C05487=1125.675,192.025,-64.166,-179.144,9.235,149.572
C05488=1125.671,192.273,-64.190,-179.142,9.238,149.572
C05489=1125.666,192.521,-64.214,-179.140,9.241,149.572
C05490=1125.662,192.771,-64.239,-179.138,9.243,149.572
C05491=1125.657,193.020,-64.262,-179.136,9.246,149.572
C05492=1125.652,193.269,-64.287,-179.135,9.248,149.572
C05493=1125.648,193.517,-64.311,-179.133,9.251,149.572
C05494=1125.644,193.766,-64.336,-179.131,9.254,149.573
C05495=1125.639,194.015,-64.360,-179.129,9.257,149.573
C05496=1125.634,194.263,-64.384,-179.127,9.259,149.573
C05497=1125.630,194.513,-64.409,-179.126,9.262,149.573
C05498=1125.625,194.761,-64.433,-179.124,9.264,149.573
C05499=1125.620,195.010,-64.458,-179.122,9.267,149.573
C05500=1125.616,195.259,-64.482,-179.121,9.269,149.573
C05501=1125.612,195.507,-64.508,-179.119,9.272,149.573
C05502=1125.607,195.755,-64.532,-179.117,9.274,149.574
C05503=1125.603,196.004,-64.556,-179.116,9.277,149.574
C05504=1125.598,196.253,-64.581,-179.114,9.279,149.574
C05505=1125.594,196.502,-64.605,-179.111,9.283,149.574
C05506=1125.589,196.751,-64.630,-179.107,9.287,149.574
C05507=1125.585,196.999,-64.654,-179.104,9.290,149.574
C05508=1125.580,197.248,-64.679,-179.099,9.295,149.574
C05509=1125.576,197.497,-64.703,-179.096,9.298,149.573
C05510=1125.571,197.745,-64.729,-179.092,9.302,149.573
C05511=1125.567,197.995,-64.754,-179.089,9.305,149.573
C05512=1125.562,198.209,-64.774,-179.086,9.308,149.573
C05513=1125.559,198.423,-64.796,-179.083,9.311,149.573
C05514=1125.555,198.637,-64.817,-179.080,9.315,149.573
C05515=1125.551,198.851,-64.839,-179.077,9.317,149.573
C05516=1125.547,199.065,-64.859,-179.074,9.320,149.573
C05517=1125.544,199.279,-64.881,-179.071,9.323,149.573
C05518=1125.540,199.492,-64.902,-179.068,9.326,149.573
C05519=1125.536,199.706,-64.923,-179.065,9.329,149.572
C05520=1125.531,199.956,-64.948,-179.062,9.332,149.572
C05521=1125.526,200.204,-64.973,-179.058,9.336,149.572
C05522=1125.523,200.453,-64.998,-179.055,9.339,149.572
C05523=1125.518,200.702,-65.023,-179.052,9.342,149.572
C05524=1125.513,200.951,-65.049,-179.048,9.345,149.572
C05525=1125.509,201.199,-65.073,-179.044,9.349,149.572
C05526=1125.505,201.448,-65.098,-179.042,9.352,149.571
C05527=1125.500,201.696,-65.123,-179.038,9.356,149.571
C05528=1125.496,201.946,-65.148,-179.035,9.358,149.571
C05529=1125.491,202.194,-65.173,-179.032,9.362,149.571
C05530=1125.487,202.443,-65.198,-179.029,9.365,149.571
C05531=1125.482,202.691,-65.223,-179.026,9.367,149.571
C05532=1125.478,202.940,-65.248,-179.022,9.371,149.571
C05533=1125.473,203.188,-65.273,-179.019,9.374,149.571
C05534=1125.469,203.438,-65.298,-179.016,9.376,149.570
C05535=1125.464,203.686,-65.324,-179.014,9.379,149.571
C05536=1125.459,203.935,-65.349,-179.010,9.383,149.570
C05537=1125.455,204.183,-65.374,-179.007,9.386,149.570
C05538=1125.451,204.432,-65.399,-179.004,9.388,149.570
C05539=1125.446,204.681,-65.424,-179.001,9.391,149.570
C05540=1125.442,204.929,-65.450,-178.999,9.394,149.570
C05541=1125.437,205.178,-65.475,-178.996,9.397,149.570
C05542=1125.432,205.427,-65.500,-178.993,9.400,149.570
C05543=1125.429,205.676,-65.525,-178.990,9.402,149.570
C05544=1125.424,205.924,-65.551,-178.988,9.406,149.570
C05545=1125.419,206.173,-65.576,-178.985,9.408,149.569
C05546=1125.415,206.422,-65.601,-178.982,9.411,149.569
C05547=1125.410,206.670,-65.627,-178.979,9.414,149.569
C05548=1125.406,206.919,-65.652,-178.976,9.417,149.569
C05549=1125.401,207.167,-65.677,-178.974,9.420,149.569
C05550=1125.397,207.416,-65.703,-178.971,9.422,149.569
C05551=1125.393,207.665,-65.729,-178.969,9.425,149.569
C05552=1125.387,207.914,-65.753,-178.966,9.428,149.569
C05553=1125.383,208.163,-65.779,-178.963,9.431,149.569
C05554=1125.379,208.411,-65.805,-178.961,9.433,149.569
C05555=1125.375,208.659,-65.830,-178.958,9.436,149.569
C05556=1125.371,208.908,-65.855,-178.956,9.439,149.569
C05557=1125.366,209.157,-65.881,-178.954,9.441,149.569
C05558=1125.361,209.406,-65.906,-178.951,9.444,149.569
C05559=1125.357,209.654,-65.932,-178.949,9.446,149.569
C05560=1125.353,209.903,-65.957,-178.947,9.450,149.569
C05561=1125.348,210.151,-65.983,-178.944,9.453,149.569
C05562=1125.344,210.400,-66.009,-178.942,9.455,149.569
C05563=1125.340,210.649,-66.034,-178.940,9.457,149.569
C05564=1125.334,210.897,-66.060,-178.937,9.460,149.569
C05565=1125.330,211.146,-66.086,-178.936,9.462,149.569
C05566=1125.326,211.395,-66.112,-178.933,9.466,149.569
C05567=1125.321,211.643,-66.137,-178.932,9.468,149.569
C05568=1125.317,211.857,-66.159,-178.930,9.471,149.569
C05569=1125.313,212.071,-66.181,-178.928,9.473,149.569
C05570=1125.310,212.285,-66.203,-178.926,9.475,149.570
C05571=1125.306,212.500,-66.225,-178.924,9.478,149.570
C05572=1125.302,212.713,-66.248,-178.923,9.480,149.570
C05573=1125.298,212.927,-66.270,-178.921,9.482,149.570
C05574=1125.295,213.140,-66.292,-178.919,9.484,149.570
C05575=1125.290,213.355,-66.314,-178.918,9.487,149.570
C05576=1125.286,213.604,-66.340,-178.916,9.489,149.570
C05577=1125.281,213.852,-66.365,-178.914,9.492,149.570
C05578=1125.277,214.100,-66.391,-178.912,9.495,149.571
C05579=1125.273,214.349,-66.416,-178.910,9.497,149.571
C05580=1125.269,214.598,-66.442,-178.909,9.500,149.571
C05581=1125.263,214.846,-66.468,-178.906,9.503,149.571
C05582=1125.259,215.095,-66.494,-178.905,9.506,149.571
C05583=1125.255,215.343,-66.520,-178.902,9.509,149.571
C05584=1125.251,215.592,-66.546,-178.900,9.511,149.571
C05585=1125.247,215.841,-66.572,-178.898,9.515,149.571
C05586=1125.242,216.089,-66.597,-178.896,9.517,149.572
C05587=1125.237,216.338,-66.624,-178.894,9.521,149.572
C05588=1125.233,216.587,-66.649,-178.892,9.523,149.572
C05589=1125.229,216.835,-66.676,-178.890,9.526,149.572
C05590=1125.224,217.084,-66.702,-178.888,9.529,149.572
C05591=1125.220,217.332,-66.727,-178.886,9.532,149.572
C05592=1125.215,217.581,-66.753,-178.883,9.535,149.572
C05593=1125.210,217.830,-66.779,-178.881,9.538,149.572
C05594=1125.206,218.078,-66.806,-178.879,9.541,149.573
C05595=1125.202,218.327,-66.831,-178.877,9.544,149.573
C05596=1125.198,218.576,-66.857,-178.874,9.547,149.573
C05597=1125.193,218.824,-66.884,-178.872,9.550,149.573
C05598=1125.189,219.073,-66.910,-178.869,9.554,149.573
C05599=1125.184,219.321,-66.935,-178.868,9.556,149.573
C05600=1125.179,219.570,-66.962,-178.865,9.559,149.573
C05601=1125.175,219.819,-66.988,-178.862,9.562,149.573
C05602=1125.171,220.067,-67.014,-178.860,9.565,149.573
C05603=1125.167,220.316,-67.040,-178.857,9.568,149.573
C05604=1125.162,220.564,-67.066,-178.855,9.571,149.573
C05605=1125.157,220.813,-67.092,-178.852,9.574,149.573
C05606=1125.154,221.061,-67.119,-178.850,9.578,149.573
C05607=1125.149,221.310,-67.145,-178.847,9.581,149.574
C05608=1125.144,221.559,-67.171,-178.845,9.584,149.574
C05609=1125.140,221.807,-67.198,-178.842,9.588,149.574
C05610=1125.135,222.056,-67.223,-178.839,9.591,149.574
C05611=1125.132,222.304,-67.250,-178.837,9.594,149.574
C05612=1125.127,222.554,-67.276,-178.834,9.597,149.574
C05613=1125.123,222.802,-67.303,-178.832,9.600,149.574
C05614=1125.118,223.050,-67.328,-178.828,9.604,149.574
C05615=1125.113,223.298,-67.355,-178.826,9.607,149.574
C05616=1125.109,223.547,-67.381,-178.823,9.610,149.574
C05617=1125.104,223.796,-67.408,-178.820,9.613,149.574
C05618=1125.100,224.044,-67.434,-178.817,9.617,149.574
C05619=1125.095,224.293,-67.461,-178.814,9.620,149.574
C05620=1125.092,224.541,-67.487,-178.811,9.624,149.574
C05621=1125.087,224.790,-67.514,-178.809,9.627,149.574
C05622=1125.083,225.038,-67.540,-178.806,9.629,149.574
C05623=1125.078,225.287,-67.567,-178.802,9.633,149.574
C05624=1125.075,225.500,-67.589,-178.800,9.636,149.574
C05625=1125.071,225.715,-67.612,-178.797,9.639,149.574
C05626=1125.067,225.928,-67.635,-178.795,9.641,149.574
C05627=1125.063,226.142,-67.658,-178.792,9.644,149.574
C05628=1125.059,226.356,-67.681,-178.790,9.647,149.574
C05629=1125.056,226.570,-67.704,-178.787,9.650,149.574
C05630=1125.052,226.784,-67.727,-178.784,9.653,149.574
C05631=1125.048,226.997,-67.750,-178.781,9.656,149.574
C05632=1125.044,227.245,-67.776,-178.778,9.659,149.574
C05633=1125.039,227.494,-67.802,-178.775,9.663,149.574
C05634=1125.034,227.743,-67.829,-178.772,9.666,149.574
C05635=1125.030,227.991,-67.856,-178.768,9.670,149.574
C05636=1125.026,228.240,-67.883,-178.765,9.672,149.573
C05637=1125.022,228.489,-67.910,-178.761,9.676,149.573
C05638=1125.017,228.738,-67.936,-178.758,9.680,149.573
C05639=1125.013,228.986,-67.963,-178.755,9.683,149.573
C05640=1125.009,229.234,-67.990,-178.752,9.686,149.573
C05641=1125.004,229.483,-68.017,-178.748,9.689,149.573
C05642=1124.999,229.731,-68.044,-178.745,9.693,149.573
C05643=1124.995,229.980,-68.070,-178.741,9.696,149.573
C05644=1124.991,230.228,-68.097,-178.737,9.700,149.572
C05645=1124.986,230.477,-68.124,-178.734,9.702,149.572
C05646=1124.982,230.725,-68.151,-178.730,9.706,149.572
C05647=1124.978,230.974,-68.178,-178.727,9.709,149.572
C05648=1124.973,231.222,-68.205,-178.724,9.712,149.572
C05649=1124.969,231.471,-68.232,-178.720,9.716,149.572
C05650=1124.965,231.719,-68.259,-178.717,9.719,149.572
C05651=1124.960,231.968,-68.286,-178.714,9.722,149.572
C05652=1124.956,232.216,-68.313,-178.711,9.725,149.571
C05653=1124.951,232.465,-68.340,-178.707,9.728,149.571
C05654=1124.947,232.714,-68.367,-178.704,9.731,149.571
C05655=1124.943,232.962,-68.394,-178.701,9.733,149.571
C05656=1124.939,233.210,-68.422,-178.697,9.737,149.571
C05657=1124.934,233.458,-68.449,-178.694,9.740,149.571
C05658=1124.930,233.708,-68.476,-178.691,9.742,149.571
C05659=1124.925,233.956,-68.503,-178.689,9.745,149.570
C05660=1124.921,234.205,-68.530,-178.685,9.749,149.570
C05661=1124.917,234.452,-68.558,-178.682,9.751,149.570
C05662=1124.912,234.701,-68.585,-178.679,9.754,149.570
C05663=1124.908,234.950,-68.612,-178.676,9.757,149.570
C05664=1124.904,235.198,-68.639,-178.673,9.760,149.570
C05665=1124.899,235.447,-68.666,-178.670,9.762,149.570
C05666=1124.895,235.695,-68.694,-178.668,9.766,149.570
C05667=1124.890,235.944,-68.721,-178.665,9.768,149.570
C05668=1124.886,236.192,-68.748,-178.662,9.771,149.570
C05669=1124.881,236.440,-68.776,-178.659,9.773,149.569
C05670=1124.877,236.689,-68.803,-178.657,9.776,149.569
C05671=1124.873,236.938,-68.831,-178.654,9.779,149.569
C05672=1124.868,237.186,-68.858,-178.651,9.781,149.569
C05673=1124.864,237.434,-68.886,-178.649,9.784,149.569
C05674=1124.861,237.683,-68.913,-178.646,9.786,149.569
C05675=1124.856,237.931,-68.940,-178.643,9.789,149.569
C05676=1124.851,238.180,-68.967,-178.641,9.791,149.569
C05677=1124.847,238.427,-68.995,-178.638,9.794,149.569
C05678=1124.842,238.677,-69.023,-178.635,9.797,149.569
C05679=1124.838,238.925,-69.051,-178.633,9.799,149.568
C05680=1124.835,239.139,-69.074,-178.631,9.801,149.569
C05681=1124.831,239.352,-69.097,-178.629,9.803,149.568
C05682=1124.828,239.566,-69.121,-178.626,9.805,149.568
C05683=1124.823,239.779,-69.145,-178.624,9.808,149.568
C05684=1124.820,239.994,-69.169,-178.622,9.810,149.568
C05685=1124.816,240.207,-69.192,-178.620,9.812,149.568
C05686=1124.812,240.421,-69.217,-178.618,9.814,149.568
C05687=1124.808,240.634,-69.240,-178.616,9.816,149.568
C05688=1124.804,240.883,-69.267,-178.614,9.818,149.568
C05689=1124.800,241.131,-69.295,-178.612,9.820,149.568
C05690=1124.795,241.379,-69.322,-178.609,9.824,149.568
C05691=1124.792,241.628,-69.350,-178.607,9.826,149.568
C05692=1124.786,241.877,-69.378,-178.605,9.828,149.568
C05693=1124.782,242.124,-69.406,-178.603,9.830,149.568
C05694=1124.778,242.373,-69.434,-178.601,9.833,149.568
C05695=1124.773,242.622,-69.461,-178.599,9.834,149.568
C05696=1124.770,242.870,-69.489,-178.596,9.838,149.568
C05697=1124.765,243.119,-69.516,-178.594,9.840,149.568
C05698=1124.761,243.367,-69.544,-178.593,9.842,149.568
C05699=1124.756,243.615,-69.573,-178.591,9.845,149.568
C05700=1124.752,243.864,-69.600,-178.589,9.847,149.568
C05701=1124.748,244.112,-69.628,-178.587,9.849,149.568
C05702=1124.743,244.360,-69.656,-178.585,9.852,149.568
C05703=1124.739,244.609,-69.683,-178.584,9.853,149.568
C05704=1124.735,244.857,-69.711,-178.582,9.855,149.569
C05705=1124.730,245.106,-69.739,-178.580,9.858,149.569
C05706=1124.726,245.354,-69.767,-178.578,9.860,149.569
C05707=1124.722,245.603,-69.795,-178.576,9.862,149.569
C05708=1124.717,245.851,-69.822,-178.575,9.865,149.569
C05709=1124.713,246.099,-69.850,-178.573,9.867,149.569
C05710=1124.708,246.347,-69.879,-178.571,9.869,149.569
C05711=1124.704,246.597,-69.906,-178.570,9.872,149.569
C05712=1124.700,246.844,-69.934,-178.568,9.874,149.569
C05713=1124.696,247.093,-69.962,-178.567,9.876,149.570
C05714=1124.691,247.341,-69.991,-178.565,9.878,149.570
C05715=1124.687,247.590,-70.019,-178.561,9.883,149.570
C05716=1124.683,247.838,-70.046,-178.555,9.887,149.569
C05717=1124.679,248.087,-70.074,-178.549,9.892,149.569
C05718=1124.674,248.335,-70.102,-178.544,9.897,149.568
C05719=1124.670,248.584,-70.130,-178.537,9.902,149.568
C05720=1124.666,248.831,-70.158,-178.532,9.906,149.567
C05721=1124.661,249.080,-70.187,-178.526,9.910,149.567
C05722=1124.657,249.328,-70.215,-178.521,9.914,149.567
C05723=1124.652,249.577,-70.243,-178.516,9.918,149.566
C05724=1124.648,249.825,-70.271,-178.512,9.922,149.566
C05725=1124.644,250.074,-70.299,-178.507,9.925,149.565
C05726=1124.639,250.322,-70.328,-178.503,9.929,149.565
C05727=1124.635,250.570,-70.356,-178.499,9.932,149.565
C05728=1124.630,250.818,-70.384,-178.495,9.935,149.565
C05729=1124.627,251.067,-70.412,-178.491,9.938,149.564
C05730=1124.622,251.315,-70.442,-178.487,9.941,149.564
C05731=1124.618,251.563,-70.470,-178.484,9.944,149.564
C05732=1124.614,251.812,-70.498,-178.480,9.946,149.564
C05733=1124.609,252.060,-70.526,-178.477,9.949,149.563
C05734=1124.606,252.309,-70.554,-178.474,9.952,149.563
C05735=1124.601,252.557,-70.583,-178.471,9.954,149.563
C05736=1124.597,252.770,-70.608,-178.469,9.956,149.563
C05737=1124.594,252.984,-70.632,-178.467,9.958,149.563
C05738=1124.590,253.197,-70.657,-178.465,9.960,149.563
C05739=1124.586,253.411,-70.681,-178.464,9.961,149.563
C05740=1124.582,253.624,-70.706,-178.462,9.963,149.563
C05741=1124.579,253.838,-70.730,-178.461,9.964,149.563
C05742=1124.575,254.052,-70.755,-178.460,9.966,149.563
C05743=1124.572,254.265,-70.780,-178.458,9.967,149.563
C05744=1124.567,254.513,-70.807,-178.457,9.969,149.563
C05745=1124.563,254.762,-70.836,-178.456,9.970,149.563
C05746=1124.559,255.010,-70.866,-178.456,9.972,149.563
C05747=1124.554,255.258,-70.893,-178.455,9.973,149.563
C05748=1124.550,255.507,-70.922,-178.455,9.974,149.564
C05749=1124.546,255.755,-70.951,-178.455,9.975,149.564
C05750=1124.541,256.003,-70.979,-178.455,9.976,149.564
C05751=1124.537,256.252,-71.008,-178.452,9.979,149.564
C05752=1124.533,256.500,-71.037,-178.449,9.982,149.564
C05753=1124.528,256.748,-71.065,-178.446,9.985,149.564
C05754=1124.524,256.997,-71.094,-178.443,9.987,149.564
C05755=1124.520,257.245,-71.123,-178.441,9.990,149.564
C05756=1124.516,257.493,-71.151,-178.437,9.994,149.564
C05757=1124.511,257.742,-71.179,-178.434,9.997,149.563
C05758=1124.507,257.990,-71.209,-178.431,9.999,149.563
C05759=1124.503,258.238,-71.237,-178.428,10.002,149.563
C05760=1124.499,258.486,-71.266,-178.425,10.005,149.563
C05761=1124.494,258.735,-71.295,-178.422,10.008,149.563
C05762=1124.491,258.983,-71.324,-178.419,10.011,149.563
C05763=1124.486,259.231,-71.352,-178.416,10.014,149.563
C05764=1124.481,259.480,-71.382,-178.413,10.017,149.563
C05765=1124.478,259.728,-71.410,-178.410,10.019,149.563
C05766=1124.474,259.976,-71.439,-178.406,10.023,149.562
C05767=1124.468,260.225,-71.468,-178.403,10.026,149.562
C05768=1124.464,260.473,-71.497,-178.400,10.028,149.562
C05769=1124.461,260.721,-71.525,-178.397,10.032,149.562
C05770=1124.456,260.970,-71.555,-178.393,10.034,149.562
C05771=1124.452,261.217,-71.584,-178.390,10.038,149.562
C05772=1124.447,261.466,-71.612,-178.387,10.041,149.562
C05773=1124.444,261.714,-71.641,-178.384,10.043,149.561
C05774=1124.439,261.963,-71.670,-178.380,10.047,149.561
C05775=1124.435,262.211,-71.699,-178.377,10.049,149.561
C05776=1124.430,262.459,-71.729,-178.373,10.052,149.561
C05777=1124.426,262.707,-71.758,-178.370,10.055,149.561
C05778=1124.422,262.956,-71.787,-178.366,10.058,149.561
C05779=1124.418,263.204,-71.816,-178.363,10.062,149.560
C05780=1124.414,263.452,-71.845,-178.359,10.064,149.560
C05781=1124.409,263.700,-71.874,-178.355,10.068,149.560
C05782=1124.405,263.949,-71.903,-178.352,10.070,149.560
C05783=1124.400,264.197,-71.932,-178.348,10.073,149.559
C05784=1124.396,264.445,-71.962,-178.344,10.077,149.559
C05785=1124.392,264.693,-71.991,-178.342,10.079,149.559
C05786=1124.388,264.942,-72.021,-178.339,10.081,149.559
C05787=1124.383,265.191,-72.049,-178.337,10.083,149.559
C05788=1124.379,265.438,-72.079,-178.334,10.086,149.559
C05789=1124.374,265.686,-72.108,-178.332,10.088,149.559
C05790=1124.370,265.935,-72.137,-178.329,10.091,149.559
C05791=1124.366,266.183,-72.167,-178.327,10.093,149.559
C05792=1124.363,266.396,-72.192,-178.324,10.095,149.558
C05793=1124.359,266.610,-72.217,-178.322,10.097,149.558
C05794=1124.355,266.823,-72.242,-178.320,10.099,149.558
C05795=1124.352,267.037,-72.268,-178.318,10.101,149.558
C05796=1124.348,267.250,-72.293,-178.316,10.103,149.558
C05797=1124.345,267.463,-72.318,-178.313,10.105,149.558
C05798=1124.341,267.677,-72.343,-178.310,10.108,149.558
C05799=1124.338,267.890,-72.368,-178.308,10.110,149.558
C05800=1124.333,268.139,-72.398,-178.306,10.112,149.558
C05801=1124.329,268.387,-72.427,-178.303,10.115,149.558
C05802=1124.325,268.635,-72.457,-178.300,10.118,149.558
C05803=1124.320,268.884,-72.487,-178.298,10.120,149.558
C05804=1124.316,269.132,-72.516,-178.295,10.123,149.557
C05805=1124.311,269.380,-72.545,-178.292,10.126,149.557
C05806=1124.307,269.627,-72.575,-178.290,10.127,149.557
C05807=1124.303,269.875,-72.605,-178.287,10.130,149.557
C05808=1124.299,270.124,-72.634,-178.284,10.133,149.557
C05809=1124.295,270.372,-72.664,-178.281,10.136,149.557
C05810=1124.291,270.620,-72.693,-178.279,10.138,149.557
C05811=1124.286,270.869,-72.723,-178.276,10.141,149.557
C05812=1124.282,271.117,-72.752,-178.273,10.143,149.557
C05813=1124.278,271.365,-72.782,-178.270,10.146,149.556
C05814=1124.273,271.613,-72.812,-178.267,10.149,149.556
C05815=1124.269,271.861,-72.842,-178.264,10.151,149.556
C05816=1124.265,272.110,-72.871,-178.261,10.153,149.556
C05817=1124.261,272.358,-72.901,-178.258,10.156,149.556
C05818=1124.257,272.606,-72.930,-178.255,10.159,149.556
C05819=1124.253,272.854,-72.960,-178.252,10.161,149.556
C05820=1124.248,273.102,-72.990,-178.249,10.164,149.556
C05821=1124.244,273.351,-73.020,-178.247,10.167,149.555
C05822=1124.240,273.599,-73.050,-178.244,10.170,149.555
C05823=1124.236,273.847,-73.080,-178.241,10.172,149.555
C05824=1124.232,274.095,-73.109,-178.237,10.175,149.555
C05825=1124.227,274.343,-73.140,-178.234,10.178,149.555
C05826=1124.223,274.592,-73.170,-178.231,10.180,149.555
C05827=1124.219,274.840,-73.199,-178.228,10.183,149.555
C05828=1124.215,275.088,-73.229,-178.226,10.186,149.555
C05829=1124.210,275.336,-73.259,-178.222,10.188,149.554
C05830=1124.206,275.584,-73.289,-178.219,10.191,149.554
C05831=1124.202,275.832,-73.319,-178.216,10.194,149.554
C05832=1124.198,276.080,-73.348,-178.213,10.197,149.554
C05833=1124.193,276.328,-73.379,-178.210,10.199,149.554
C05834=1124.190,276.577,-73.409,-178.207,10.202,149.554
C05835=1124.186,276.825,-73.439,-178.204,10.205,149.553
C05836=1124.181,277.074,-73.469,-178.200,10.208,149.553
C05837=1124.177,277.321,-73.499,-178.197,10.211,149.553
C05838=1124.173,277.569,-73.529,-178.194,10.213,149.553
C05839=1124.168,277.817,-73.559,-178.191,10.216,149.553
C05840=1124.164,278.066,-73.589,-178.188,10.218,149.553
C05841=1124.161,278.314,-73.619,-178.185,10.221,149.552
C05842=1124.156,278.563,-73.650,-178.181,10.224,149.552
C05843=1124.152,278.810,-73.680,-178.178,10.227,149.552
C05844=1124.148,279.058,-73.710,-178.175,10.230,149.552
C05845=1124.143,279.306,-73.740,-178.171,10.232,149.552
C05846=1124.139,279.554,-73.770,-178.169,10.235,149.552
C05847=1124.135,279.803,-73.801,-178.165,10.238,149.551
C05848=1124.132,280.016,-73.826,-178.162,10.240,149.551
C05849=1124.128,280.229,-73.853,-178.159,10.242,149.551
C05850=1124.125,280.442,-73.879,-178.156,10.245,149.551
C05851=1124.120,280.656,-73.905,-178.154,10.247,149.551
C05852=1124.118,280.869,-73.931,-178.150,10.249,149.550
C05853=1124.114,281.082,-73.957,-178.147,10.252,149.550
C05854=1124.110,281.296,-73.982,-178.144,10.255,149.550
C05855=1124.106,281.509,-74.009,-178.142,10.257,149.550
C05856=1124.102,281.757,-74.039,-178.138,10.259,149.550
C05857=1124.098,282.005,-74.070,-178.135,10.262,149.549
C05858=1124.094,282.253,-74.100,-178.133,10.265,149.549
C05859=1124.089,282.502,-74.130,-178.129,10.267,149.549
C05860=1124.085,282.749,-74.161,-178.126,10.270,149.549
C05861=1124.082,282.998,-74.192,-178.123,10.272,149.549
C05862=1124.077,283.246,-74.223,-178.120,10.275,149.549
C05863=1124.073,283.493,-74.253,-178.118,10.277,149.549
C05864=1124.068,283.741,-74.283,-178.114,10.279,149.548
C05865=1124.065,283.990,-74.314,-178.111,10.282,149.548
C05866=1124.061,284.238,-74.345,-178.108,10.285,149.548
C05867=1124.056,284.486,-74.375,-178.105,10.287,149.548
C05868=1124.052,284.735,-74.405,-178.102,10.290,149.547
C05869=1124.048,284.983,-74.436,-178.099,10.292,149.547
C05870=1124.043,285.231,-74.467,-178.096,10.295,149.547
C05871=1124.039,285.478,-74.497,-178.093,10.298,149.547
C05872=1124.035,285.727,-74.528,-178.090,10.300,149.547
C05873=1124.031,285.975,-74.559,-178.087,10.302,149.547
C05874=1124.027,286.222,-74.589,-178.084,10.305,149.547
C05875=1124.023,286.471,-74.620,-178.081,10.307,149.546
C05876=1124.018,286.719,-74.651,-178.078,10.310,149.546
C05877=1124.014,286.967,-74.681,-178.075,10.313,149.546
C05878=1124.011,287.215,-74.713,-178.071,10.315,149.546
C05879=1124.006,287.463,-74.744,-178.068,10.318,149.546
C05880=1124.003,287.711,-74.774,-178.065,10.320,149.545
C05881=1123.998,287.959,-74.805,-178.062,10.323,149.545
C05882=1123.993,288.207,-74.836,-178.059,10.325,149.545
C05883=1123.989,288.456,-74.867,-178.057,10.328,149.545
C05884=1123.986,288.703,-74.897,-178.053,10.330,149.545
C05885=1123.981,288.951,-74.928,-178.050,10.333,149.545
C05886=1123.977,289.199,-74.960,-178.047,10.335,149.544
C05887=1123.973,289.447,-74.991,-178.044,10.338,149.544
C05888=1123.969,289.696,-75.021,-178.041,10.341,149.544
C05889=1123.965,289.944,-75.052,-178.038,10.343,149.544
C05890=1123.960,290.191,-75.083,-178.035,10.346,149.544
C05891=1123.956,290.440,-75.114,-178.031,10.348,149.543
C05892=1123.952,290.687,-75.145,-178.029,10.351,149.543
C05893=1123.948,290.936,-75.176,-178.026,10.353,149.543
C05894=1123.944,291.183,-75.207,-178.023,10.355,149.543
C05895=1123.940,291.432,-75.238,-178.020,10.358,149.543
C05896=1123.936,291.680,-75.269,-178.017,10.361,149.543
C05897=1123.932,291.928,-75.301,-178.013,10.363,149.542
C05898=1123.927,292.176,-75.332,-178.010,10.366,149.542
C05899=1123.923,292.424,-75.363,-178.007,10.369,149.542
C05900=1123.919,292.672,-75.394,-178.004,10.371,149.542
C05901=1123.916,292.920,-75.425,-178.001,10.374,149.542
C05902=1123.911,293.167,-75.456,-177.998,10.376,149.542
C05903=1123.907,293.415,-75.487,-177.995,10.378,149.541
C05904=1123.903,293.629,-75.514,-177.992,10.381,149.541
C05905=1123.900,293.842,-75.541,-177.990,10.383,149.541
C05906=1123.896,294.056,-75.568,-177.987,10.385,149.541
C05907=1123.893,294.268,-75.595,-177.985,10.387,149.541
C05908=1123.889,294.482,-75.622,-177.982,10.389,149.541
C05909=1123.885,294.695,-75.649,-177.979,10.392,149.540
C05910=1123.882,294.907,-75.675,-177.977,10.394,149.540
C05911=1123.879,295.121,-75.702,-177.974,10.395,149.540
C05912=1123.875,295.368,-75.734,-177.971,10.398,149.540
C05913=1123.870,295.617,-75.765,-177.968,10.401,149.540
C05914=1123.867,295.865,-75.797,-177.965,10.403,149.540
C05915=1123.862,296.112,-75.828,-177.962,10.406,149.540
C05916=1123.858,296.361,-75.859,-177.958,10.409,149.539
C05917=1123.854,296.608,-75.891,-177.956,10.411,149.539
C05918=1123.849,296.857,-75.922,-177.952,10.414,149.539
C05919=1123.845,297.105,-75.954,-177.949,10.417,149.539
C05920=1123.841,297.353,-75.986,-177.946,10.419,149.539
C05921=1123.837,297.601,-76.016,-177.944,10.421,149.538
C05922=1123.833,297.849,-76.048,-177.940,10.423,149.538
C05923=1123.829,298.097,-76.080,-177.937,10.426,149.538
C05924=1123.825,298.345,-76.111,-177.934,10.429,149.538
C05925=1123.821,298.593,-76.143,-177.931,10.431,149.538
C05926=1123.817,298.840,-76.174,-177.928,10.434,149.537
C05927=1123.813,299.088,-76.206,-177.925,10.437,149.537
C05928=1123.809,299.337,-76.237,-177.922,10.439,149.537
C05929=1123.804,299.584,-76.269,-177.919,10.442,149.537
C05930=1123.800,299.832,-76.301,-177.915,10.444,149.537
C05931=1123.797,300.080,-76.333,-177.912,10.447,149.537
C05932=1123.792,300.328,-76.364,-177.910,10.449,149.536
C05933=1123.788,300.576,-76.396,-177.907,10.451,149.536
C05934=1123.784,300.824,-76.427,-177.903,10.454,149.536
C05935=1123.779,301.072,-76.459,-177.900,10.457,149.536
C05936=1123.776,301.320,-76.491,-177.897,10.459,149.536
C05937=1123.771,301.567,-76.523,-177.894,10.462,149.536
C05938=1123.768,301.816,-76.555,-177.891,10.464,149.535
C05939=1123.763,302.064,-76.587,-177.887,10.467,149.535
C05940=1123.759,302.311,-76.619,-177.885,10.469,149.535
C05941=1123.755,302.560,-76.650,-177.881,10.472,149.535
C05942=1123.751,302.808,-76.682,-177.878,10.475,149.535
C05943=1123.746,303.056,-76.714,-177.875,10.477,149.534
C05944=1123.743,303.304,-76.745,-177.873,10.479,149.534
C05945=1123.739,303.552,-76.777,-177.869,10.481,149.534
C05946=1123.734,303.799,-76.809,-177.866,10.484,149.534
C05947=1123.730,304.047,-76.841,-177.863,10.487,149.534
C05948=1123.726,304.295,-76.873,-177.860,10.489,149.534
C05949=1123.722,304.543,-76.906,-177.857,10.492,149.533
C05950=1123.718,304.790,-76.938,-177.854,10.495,149.533
C05951=1123.714,305.038,-76.970,-177.851,10.497,149.533
C05952=1123.710,305.287,-77.002,-177.848,10.500,149.533
C05953=1123.706,305.535,-77.034,-177.844,10.502,149.533
C05954=1123.702,305.782,-77.065,-177.841,10.505,149.533
C05955=1123.697,306.031,-77.098,-177.838,10.507,149.532
C05956=1123.694,306.279,-77.130,-177.835,10.510,149.532
C05957=1123.689,306.527,-77.162,-177.832,10.512,149.532
C05958=1123.685,306.774,-77.194,-177.829,10.514,149.532
C05959=1123.681,307.022,-77.226,-177.826,10.517,149.532
C05960=1123.678,307.235,-77.254,-177.823,10.519,149.531
C05961=1123.674,307.448,-77.281,-177.820,10.521,149.531
C05962=1123.671,307.661,-77.309,-177.818,10.523,149.531
C05963=1123.667,307.874,-77.337,-177.815,10.526,149.531
C05964=1123.663,308.087,-77.364,-177.813,10.528,149.531
C05965=1123.660,308.300,-77.392,-177.810,10.531,149.531
C05966=1123.656,308.514,-77.420,-177.807,10.532,149.530
C05967=1123.653,308.726,-77.447,-177.805,10.534,149.530
C05968=1123.649,308.973,-77.480,-177.802,10.537,149.530
C05969=1123.645,309.222,-77.512,-177.798,10.540,149.530
C05970=1123.641,309.470,-77.544,-177.795,10.542,149.530
C05971=1123.637,309.718,-77.577,-177.792,10.545,149.530
C05972=1123.633,309.965,-77.609,-177.789,10.547,149.529
C05973=1123.629,310.213,-77.642,-177.786,10.550,149.529
C05974=1123.625,310.461,-77.674,-177.783,10.552,149.529
C05975=1123.620,310.709,-77.706,-177.780,10.555,149.529
C05976=1123.617,310.956,-77.739,-177.776,10.558,149.529
C05977=1123.613,311.205,-77.771,-177.774,10.559,149.528
C05978=1123.608,311.453,-77.804,-177.771,10.562,149.528
C05979=1123.604,311.700,-77.836,-177.767,10.564,149.528
C05980=1123.600,311.948,-77.869,-177.764,10.567,149.528
C05981=1123.596,312.196,-77.901,-177.761,10.570,149.528
C05982=1123.592,312.443,-77.934,-177.758,10.572,149.528
C05983=1123.588,312.692,-77.967,-177.755,10.575,149.527
C05984=1123.584,312.939,-77.999,-177.751,10.577,149.527
C05985=1123.580,313.187,-78.032,-177.749,10.580,149.527
C05986=1123.577,313.435,-78.064,-177.745,10.583,149.527
C05987=1123.572,313.683,-78.097,-177.742,10.585,149.527
C05988=1123.568,313.931,-78.130,-177.739,10.588,149.527
C05989=1123.565,314.178,-78.162,-177.736,10.590,149.526
C05990=1123.560,314.427,-78.195,-177.733,10.593,149.526
C05991=1123.555,314.674,-78.227,-177.730,10.595,149.526
C05992=1123.552,314.922,-78.259,-177.727,10.597,149.526
C05993=1123.547,315.170,-78.292,-177.724,10.600,149.526
C05994=1123.543,315.417,-78.326,-177.720,10.602,149.525
C05995=1123.540,315.665,-78.357,-177.717,10.605,149.525
C05996=1123.536,315.913,-78.391,-177.714,10.607,149.525
C05997=1123.531,316.161,-78.424,-177.711,10.610,149.525
C05998=1123.527,316.409,-78.457,-177.708,10.613,149.525
C05999=1123.524,316.657,-78.489,-177.705,10.615,149.524
C06000=1123.519,316.904,-78.522,-177.702,10.618,149.524
C06001=1123.515,317.152,-78.555,-177.698,10.620,149.524
C06002=1123.511,317.400,-78.588,-177.695,10.623,149.524
C06003=1123.508,317.647,-78.621,-177.692,10.626,149.524
C06004=1123.503,317.896,-78.653,-177.689,10.628,149.524
C06005=1123.499,318.143,-78.686,-177.686,10.630,149.523
C06006=1123.495,318.391,-78.720,-177.683,10.632,149.523
C06007=1123.491,318.639,-78.753,-177.680,10.635,149.523
C06008=1123.488,318.887,-78.786,-177.677,10.638,149.523
C06009=1123.484,319.135,-78.819,-177.674,10.640,149.523
C06010=1123.480,319.382,-78.852,-177.670,10.643,149.522
C06011=1123.475,319.631,-78.884,-177.667,10.645,149.522
C06012=1123.471,319.878,-78.918,-177.664,10.648,149.522
C06013=1123.467,320.126,-78.951,-177.661,10.651,149.522
C06014=1123.463,320.374,-78.984,-177.658,10.653,149.522
C06015=1123.460,320.621,-79.016,-177.654,10.655,149.521
C06016=1123.456,320.834,-79.045,-177.652,10.657,149.521
C06017=1123.452,321.047,-79.074,-177.649,10.660,149.521
C06018=1123.450,321.260,-79.102,-177.646,10.662,149.521
C06019=1123.446,321.473,-79.131,-177.644,10.664,149.521
C06020=1123.442,321.685,-79.159,-177.641,10.666,149.521
C06021=1123.439,321.898,-79.187,-177.639,10.668,149.521
C06022=1123.435,322.111,-79.216,-177.636,10.670,149.520
C06023=1123.432,322.324,-79.245,-177.633,10.673,149.520
C06024=1123.428,322.571,-79.278,-177.630,10.675,149.520
C06025=1123.424,322.819,-79.312,-177.627,10.678,149.520
C06026=1123.420,323.067,-79.345,-177.623,10.680,149.520
C06027=1123.416,323.315,-79.378,-177.620,10.683,149.519
C06028=1123.412,323.563,-79.411,-177.618,10.685,149.519
C06029=1123.408,323.811,-79.445,-177.614,10.687,149.519
C06030=1123.404,324.058,-79.478,-177.611,10.690,149.519
C06031=1123.400,324.305,-79.512,-177.608,10.693,149.519
C06032=1123.396,324.553,-79.545,-177.605,10.695,149.519
C06033=1123.392,324.802,-79.578,-177.602,10.697,149.518
C06034=1123.388,325.049,-79.611,-177.599,10.700,149.518
C06035=1123.384,325.296,-79.645,-177.595,10.703,149.518
C06036=1123.380,325.544,-79.678,-177.592,10.705,149.518
C06037=1123.376,325.792,-79.712,-177.589,10.708,149.518
C06038=1123.372,326.040,-79.745,-177.586,10.710,149.517
C06039=1123.368,326.287,-79.779,-177.582,10.713,149.517
C06040=1123.364,326.535,-79.812,-177.579,10.716,149.517
C06041=1123.360,326.783,-79.845,-177.576,10.718,149.517
C06042=1123.356,327.030,-79.879,-177.573,10.720,149.517
C06043=1123.352,327.279,-79.913,-177.571,10.722,149.517
C06044=1123.348,327.527,-79.946,-177.567,10.725,149.516
C06045=1123.344,327.774,-79.980,-177.564,10.727,149.516
C06046=1123.340,328.021,-80.013,-177.561,10.730,149.516
C06047=1123.336,328.268,-80.047,-177.558,10.733,149.516
C06048=1123.333,328.517,-80.081,-177.554,10.735,149.516
C06049=1123.328,328.765,-80.115,-177.551,10.737,149.515
C06050=1123.324,329.012,-80.148,-177.548,10.740,149.515
C06051=1123.320,329.260,-80.182,-177.545,10.743,149.515
C06052=1123.317,329.508,-80.216,-177.541,10.745,149.515
C06053=1123.312,329.755,-80.249,-177.539,10.748,149.515
C06054=1123.308,330.003,-80.283,-177.535,10.750,149.514
C06055=1123.304,330.251,-80.317,-177.532,10.753,149.514
C06056=1123.300,330.498,-80.351,-177.529,10.755,149.514
C06057=1123.297,330.745,-80.385,-177.526,10.758,149.514
C06058=1123.292,330.993,-80.418,-177.522,10.760,149.514
C06059=1123.288,331.241,-80.453,-177.520,10.762,149.513
C06060=1123.284,331.489,-80.486,-177.517,10.765,149.513
C06061=1123.281,331.736,-80.520,-177.513,10.767,149.513
C06062=1123.277,331.984,-80.555,-177.510,10.770,149.513
C06063=1123.272,332.232,-80.588,-177.507,10.772,149.513
C06064=1123.269,332.479,-80.622,-177.504,10.775,149.513
C06065=1123.264,332.728,-80.656,-177.501,10.777,149.512
C06066=1123.260,332.975,-80.690,-177.497,10.780,149.512
C06067=1123.257,333.222,-80.723,-177.494,10.782,149.512
C06068=1123.253,333.470,-80.758,-177.491,10.785,149.512
C06069=1123.249,333.718,-80.791,-177.488,10.788,149.511
C06070=1123.245,333.966,-80.826,-177.484,10.790,149.511
C06071=1123.241,334.213,-80.860,-177.481,10.793,149.511
C06072=1123.237,334.426,-80.889,-177.479,10.795,149.511
C06073=1123.234,334.638,-80.919,-177.476,10.796,149.511
C06074=1123.230,334.851,-80.948,-177.473,10.799,149.511
C06075=1123.227,335.063,-80.977,-177.470,10.801,149.510
C06076=1123.224,335.276,-81.006,-177.467,10.803,149.510
C06077=1123.221,335.488,-81.036,-177.465,10.805,149.510
C06078=1123.218,335.702,-81.065,-177.463,10.807,149.510
C06079=1123.214,335.914,-81.094,-177.459,10.810,149.510
C06080=1123.210,336.162,-81.128,-177.456,10.812,149.510
C06081=1123.206,336.410,-81.162,-177.453,10.815,149.509
C06082=1123.202,336.658,-81.197,-177.450,10.817,149.509
C06083=1123.198,336.905,-81.231,-177.446,10.820,149.509
C06084=1123.194,337.153,-81.266,-177.444,10.822,149.509
C06085=1123.190,337.400,-81.299,-177.441,10.824,149.509
C06086=1123.186,337.648,-81.334,-177.437,10.827,149.508
C06087=1123.182,337.895,-81.368,-177.434,10.829,149.508
C06088=1123.178,338.143,-81.403,-177.431,10.832,149.508
C06089=1123.174,338.390,-81.437,-177.428,10.834,149.508
C06090=1123.171,338.639,-81.472,-177.425,10.837,149.508
C06091=1123.167,338.886,-81.506,-177.421,10.839,149.507
C06092=1123.162,339.133,-81.540,-177.418,10.842,149.507
C06093=1123.158,339.381,-81.575,-177.415,10.844,149.507
C06094=1123.154,339.628,-81.609,-177.412,10.847,149.507
C06095=1123.150,339.876,-81.644,-177.408,10.849,149.507
C06096=1123.147,340.123,-81.677,-177.405,10.852,149.506
C06097=1123.143,340.372,-81.712,-177.402,10.854,149.506
C06098=1123.138,340.618,-81.747,-177.399,10.857,149.506
C06099=1123.135,340.866,-81.782,-177.395,10.860,149.506
C06100=1123.130,341.114,-81.816,-177.392,10.862,149.506
C06101=1123.127,341.362,-81.851,-177.389,10.864,149.505
C06102=1123.123,341.609,-81.885,-177.386,10.866,149.505
C06103=1123.119,341.857,-81.920,-177.383,10.869,149.505
C06104=1123.115,342.104,-81.955,-177.380,10.871,149.505
C06105=1123.111,342.352,-81.989,-177.377,10.874,149.505
C06106=1123.107,342.600,-82.024,-177.373,10.876,149.504
C06107=1123.103,342.847,-82.058,-177.370,10.879,149.504
C06108=1123.100,343.094,-82.093,-177.367,10.881,149.504
C06109=1123.095,343.342,-82.128,-177.364,10.884,149.504
C06110=1123.091,343.590,-82.163,-177.360,10.886,149.504
C06111=1123.088,343.836,-82.197,-177.357,10.889,149.503
C06112=1123.084,344.084,-82.232,-177.354,10.891,149.503
C06113=1123.080,344.333,-82.267,-177.350,10.894,149.503
C06114=1123.075,344.579,-82.302,-177.348,10.897,149.503
C06115=1123.072,344.827,-82.336,-177.344,10.899,149.503
C06116=1123.066,345.174,-82.386,-177.340,10.902,149.502
C06117=1123.061,345.520,-82.434,-177.335,10.906,149.502
C06118=1123.055,345.866,-82.483,-177.331,10.909,149.502
C06119=1123.050,346.212,-82.532,-177.326,10.913,149.501
C06120=1123.045,346.459,-82.566,-177.323,10.915,149.501
C06121=1123.042,346.707,-82.602,-177.320,10.918,149.501
C06122=1123.039,346.955,-82.636,-177.317,10.920,149.501
C06123=1123.034,347.202,-82.671,-177.314,10.922,149.501
C06124=1123.030,347.450,-82.706,-177.311,10.924,149.500
C06125=1123.027,347.697,-82.742,-177.307,10.927,149.500
C06126=1123.022,347.945,-82.776,-177.304,10.929,149.500
C06127=1123.018,348.192,-82.812,-177.301,10.932,149.500
C06128=1123.013,348.518,-82.858,-177.297,10.935,149.500
C06129=1123.008,348.845,-82.903,-177.292,10.939,149.499
C06130=1123.003,349.172,-82.950,-177.288,10.942,149.499
C06131=1122.998,349.498,-82.997,-177.284,10.945,149.499
C06132=1122.994,349.746,-83.031,-177.280,10.948,149.499
C06133=1122.990,349.993,-83.067,-177.276,10.951,149.498
C06134=1122.986,350.240,-83.102,-177.273,10.953,149.498
C06135=1122.983,350.488,-83.138,-177.270,10.955,149.498
C06136=1122.979,350.736,-83.173,-177.266,10.958,149.498
C06137=1122.975,350.982,-83.208,-177.262,10.961,149.497
C06138=1122.971,351.230,-83.243,-177.259,10.964,149.497
C06139=1122.967,351.477,-83.279,-177.256,10.966,149.497
C06140=1122.963,351.726,-83.314,-177.252,10.968,149.496
C06141=1122.959,351.972,-83.349,-177.248,10.971,149.496
C06142=1122.955,352.220,-83.384,-177.245,10.974,149.496
C06143=1122.952,352.467,-83.420,-177.241,10.976,149.496
C06144=1122.948,352.715,-83.455,-177.238,10.979,149.496
C06145=1122.944,352.962,-83.491,-177.234,10.981,149.495
C06146=1122.940,353.210,-83.525,-177.230,10.984,149.495
C06147=1122.936,353.457,-83.561,-177.227,10.987,149.495
C06148=1122.932,353.705,-83.597,-177.224,10.989,149.495
C06149=1122.929,353.952,-83.632,-177.220,10.992,149.494
C06150=1122.924,354.199,-83.668,-177.217,10.994,149.494
C06151=1122.920,354.447,-83.703,-177.213,10.996,149.494
C06152=1122.916,354.694,-83.739,-177.210,10.999,149.494
C06153=1122.913,354.942,-83.775,-177.206,11.002,149.493
C06154=1122.909,355.189,-83.810,-177.203,11.004,149.493
C06155=1122.906,355.437,-83.846,-177.199,11.007,149.493
C06156=1122.901,355.684,-83.881,-177.196,11.009,149.492
C06157=1122.898,355.931,-83.916,-177.193,11.011,149.492
C06158=1122.893,356.179,-83.953,-177.189,11.014,149.492
C06159=1122.890,356.427,-83.988,-177.186,11.016,149.492
C06160=1122.886,356.674,-84.024,-177.182,11.019,149.491
C06161=1122.882,356.921,-84.060,-177.178,11.022,149.491
C06162=1122.879,357.168,-84.095,-177.175,11.024,149.491
C06163=1122.874,357.416,-84.132,-177.172,11.027,149.491
C06164=1122.871,357.664,-84.167,-177.168,11.029,149.490
C06165=1122.867,357.910,-84.202,-177.165,11.031,149.490
C06166=1122.863,358.158,-84.238,-177.161,11.034,149.490
C06167=1122.859,358.405,-84.274,-177.158,11.036,149.490
C06168=1122.855,358.653,-84.310,-177.154,11.038,149.489
C06169=1122.851,358.900,-84.346,-177.151,11.041,149.489
C06170=1122.848,359.148,-84.381,-177.148,11.043,149.489
C06171=1122.844,359.395,-84.418,-177.144,11.046,149.489
C06172=1122.840,359.642,-84.454,-177.141,11.048,149.488
C06173=1122.836,359.890,-84.489,-177.137,11.050,149.488
C06174=1122.833,360.137,-84.525,-177.134,11.053,149.488
C06175=1122.829,360.385,-84.562,-177.131,11.055,149.488
C06176=1122.825,360.632,-84.597,-177.127,11.057,149.487
C06177=1122.821,360.880,-84.633,-177.124,11.060,149.487
C06178=1122.817,361.127,-84.670,-177.121,11.062,149.487
C06179=1122.814,361.374,-84.705,-177.117,11.065,149.487
C06180=1122.810,361.586,-84.736,-177.114,11.067,149.486
C06181=1122.807,361.799,-84.767,-177.111,11.069,149.486
C06182=1122.804,362.012,-84.799,-177.108,11.071,149.486
C06183=1122.800,362.223,-84.830,-177.105,11.073,149.486
C06184=1122.798,362.436,-84.860,-177.103,11.075,149.485
C06185=1122.794,362.648,-84.891,-177.099,11.077,149.485
C06186=1122.791,362.860,-84.922,-177.097,11.079,149.485
C06187=1122.787,363.073,-84.953,-177.094,11.082,149.485
C06188=1122.783,363.320,-84.990,-177.090,11.084,149.484
C06189=1122.780,363.568,-85.026,-177.087,11.086,149.484
C06190=1122.777,363.815,-85.062,-177.084,11.088,149.484
C06191=1122.773,364.062,-85.099,-177.081,11.091,149.484
C06192=1122.769,364.310,-85.134,-177.077,11.093,149.484
C06193=1122.765,364.557,-85.171,-177.074,11.095,149.483
C06194=1122.761,364.805,-85.206,-177.070,11.098,149.483
C06195=1122.757,365.052,-85.243,-177.067,11.100,149.483
C06196=1122.754,365.299,-85.280,-177.064,11.103,149.483
C06197=1122.749,365.546,-85.316,-177.061,11.105,149.482
C06198=1122.746,365.793,-85.352,-177.057,11.108,149.482
C06199=1122.742,366.041,-85.389,-177.054,11.110,149.482
C06200=1122.738,366.288,-85.424,-177.050,11.112,149.481
C06201=1122.734,366.535,-85.461,-177.047,11.115,149.481
C06202=1122.731,366.782,-85.498,-177.044,11.116,149.481
C06203=1122.727,367.031,-85.534,-177.041,11.119,149.481
C06204=1122.723,367.278,-85.571,-177.038,11.121,149.481
C06205=1122.719,367.525,-85.607,-177.034,11.124,149.480
C06206=1122.715,367.772,-85.644,-177.031,11.126,149.480
C06207=1122.712,368.019,-85.680,-177.028,11.129,149.480
C06208=1122.708,368.267,-85.716,-177.024,11.131,149.480
C06209=1122.704,368.514,-85.753,-177.021,11.133,149.479
C06210=1122.700,368.761,-85.790,-177.017,11.136,149.479
C06211=1122.697,369.009,-85.827,-177.015,11.138,149.479
C06212=1122.693,369.256,-85.862,-177.011,11.140,149.479
C06213=1122.689,369.503,-85.899,-177.008,11.142,149.478
C06214=1122.685,369.750,-85.936,-177.005,11.145,149.478
C06215=1122.681,369.997,-85.972,-177.002,11.147,149.478
C06216=1122.677,370.245,-86.009,-176.998,11.150,149.478
C06217=1122.674,370.492,-86.046,-176.995,11.152,149.478
C06218=1122.670,370.740,-86.083,-176.992,11.154,149.477
C06219=1122.666,370.986,-86.120,-176.989,11.157,149.477
C06220=1122.662,371.234,-86.156,-176.986,11.159,149.477
C06221=1122.658,371.481,-86.193,-176.982,11.162,149.477
C06222=1122.655,371.728,-86.230,-176.979,11.164,149.477
C06223=1122.651,371.976,-86.267,-176.976,11.166,149.476
C06224=1122.647,372.223,-86.304,-176.973,11.168,149.476
C06225=1122.643,372.470,-86.340,-176.970,11.171,149.476
C06226=1122.640,372.718,-86.377,-176.967,11.173,149.476
C06227=1122.636,372.965,-86.414,-176.963,11.176,149.476
C06228=1122.632,373.212,-86.451,-176.960,11.178,149.475
C06229=1122.628,373.459,-86.488,-176.957,11.181,149.475
C06230=1122.625,373.707,-86.524,-176.954,11.183,149.475
C06231=1122.621,373.954,-86.561,-176.951,11.185,149.475
C06232=1122.618,374.201,-86.599,-176.948,11.188,149.475
C06233=1122.613,374.448,-86.636,-176.944,11.190,149.474
C06234=1122.610,374.696,-86.673,-176.941,11.193,149.474
C06235=1122.607,374.942,-86.709,-176.938,11.194,149.474
C06236=1122.603,375.155,-86.742,-176.936,11.197,149.474
C06237=1122.599,375.367,-86.773,-176.933,11.199,149.474
C06238=1122.597,375.579,-86.805,-176.931,11.201,149.474
C06239=1122.593,375.792,-86.836,-176.928,11.202,149.473
C06240=1122.590,376.004,-86.868,-176.925,11.205,149.473
C06241=1122.587,376.216,-86.900,-176.922,11.207,149.473
C06242=1122.583,376.428,-86.932,-176.920,11.209,149.473
C06243=1122.580,376.640,-86.964,-176.917,11.211,149.473
C06244=1122.576,376.887,-87.001,-176.914,11.213,149.473
C06245=1122.573,377.135,-87.038,-176.911,11.216,149.473
C06246=1122.569,377.382,-87.076,-176.908,11.218,149.472
C06247=1122.565,377.629,-87.112,-176.905,11.221,149.472
C06248=1122.561,377.877,-87.150,-176.902,11.223,149.472
C06249=1122.558,378.123,-87.187,-176.899,11.225,149.472
C06250=1122.554,378.370,-87.223,-176.896,11.228,149.472
C06251=1122.551,378.618,-87.261,-176.893,11.231,149.472
C06252=1122.547,378.865,-87.298,-176.890,11.233,149.472
C06253=1122.543,379.112,-87.335,-176.887,11.235,149.472
C06254=1122.540,379.359,-87.373,-176.884,11.238,149.471
C06255=1122.536,379.606,-87.410,-176.881,11.240,149.471
C06256=1122.532,379.854,-87.448,-176.878,11.243,149.471
C06257=1122.528,380.101,-87.485,-176.875,11.245,149.471
C06258=1122.525,380.347,-87.522,-176.872,11.248,149.471
C06259=1122.521,380.595,-87.560,-176.869,11.250,149.471
C06260=1122.517,380.842,-87.597,-176.866,11.253,149.471
C06261=1122.512,381.089,-87.635,-176.863,11.255,149.470
C06262=1122.509,381.337,-87.672,-176.861,11.257,149.470
C06263=1122.505,381.584,-87.709,-176.857,11.260,149.470
C06264=1122.502,381.831,-87.747,-176.854,11.263,149.470
C06265=1122.498,382.078,-87.784,-176.851,11.265,149.470
C06266=1122.495,382.326,-87.822,-176.849,11.267,149.470
C06267=1122.491,382.572,-87.860,-176.846,11.270,149.470
C06268=1122.487,382.819,-87.897,-176.843,11.273,149.470
C06269=1122.484,383.067,-87.934,-176.840,11.275,149.470
C06270=1122.480,383.313,-87.972,-176.837,11.277,149.470
C06271=1122.476,383.561,-88.009,-176.835,11.280,149.470
C06272=1122.473,383.808,-88.047,-176.833,11.282,149.470
C06273=1122.469,384.055,-88.085,-176.831,11.284,149.470
C06274=1122.464,384.302,-88.122,-176.829,11.286,149.470
C06275=1122.461,384.550,-88.160,-176.827,11.288,149.470
C06276=1122.458,384.796,-88.198,-176.825,11.291,149.470
C06277=1122.454,385.044,-88.235,-176.824,11.292,149.470
C06278=1122.450,385.291,-88.273,-176.821,11.294,149.470
C06279=1122.447,385.538,-88.310,-176.820,11.296,149.470
C06280=1122.443,385.785,-88.349,-176.818,11.299,149.470
C06281=1122.439,386.033,-88.386,-176.816,11.301,149.470
C06282=1122.435,386.279,-88.423,-176.815,11.303,149.470
C06283=1122.431,386.526,-88.461,-176.812,11.305,149.470
C06284=1122.428,386.773,-88.499,-176.810,11.307,149.471
C06285=1122.424,387.021,-88.537,-176.809,11.310,149.471
C06286=1122.420,387.268,-88.574,-176.807,11.312,149.471
C06287=1122.417,387.515,-88.612,-176.805,11.315,149.471
C06288=1122.413,387.762,-88.650,-176.803,11.317,149.471
C06289=1122.410,388.009,-88.688,-176.801,11.319,149.471
C06290=1122.406,388.256,-88.726,-176.800,11.321,149.471
C06291=1122.402,388.503,-88.764,-176.798,11.323,149.472
C06292=1122.400,388.715,-88.796,-176.796,11.326,149.472
C06293=1122.396,388.928,-88.828,-176.796,11.327,149.472
C06294=1122.393,389.140,-88.861,-176.794,11.330,149.472
C06295=1122.389,389.351,-88.893,-176.792,11.331,149.472
C06296=1122.386,389.564,-88.925,-176.791,11.334,149.473
C06297=1122.383,389.775,-88.958,-176.790,11.336,149.473
C06298=1122.380,389.987,-88.991,-176.788,11.338,149.473
C06299=1122.376,390.200,-89.023,-176.787,11.340,149.473
C06300=1122.373,390.447,-89.061,-176.786,11.343,149.473
C06301=1122.370,390.694,-89.099,-176.784,11.345,149.473
C06302=1122.366,390.941,-89.137,-176.782,11.348,149.474
C06303=1122.362,391.188,-89.175,-176.781,11.350,149.474
C06304=1122.359,391.435,-89.213,-176.779,11.353,149.474
C06305=1122.355,391.682,-89.251,-176.777,11.355,149.475
C06306=1122.351,391.929,-89.289,-176.776,11.358,149.475
C06307=1122.348,392.176,-89.327,-176.774,11.361,149.475
C06308=1122.345,392.424,-89.365,-176.772,11.364,149.476
C06309=1122.340,392.670,-89.403,-176.771,11.367,149.476
C06310=1122.337,392.918,-89.441,-176.769,11.370,149.476
C06311=1122.333,393.164,-89.478,-176.768,11.372,149.477
C06312=1122.329,393.412,-89.517,-176.766,11.375,149.477
C06313=1122.325,393.658,-89.555,-176.765,11.378,149.477
C06314=1122.322,393.906,-89.592,-176.764,11.381,149.478
C06315=1122.318,394.153,-89.631,-176.762,11.383,149.478
C06316=1122.314,394.400,-89.669,-176.761,11.386,149.478
C06317=1122.310,394.647,-89.707,-176.760,11.389,149.479
C06318=1122.307,394.894,-89.745,-176.758,11.392,149.479
C06319=1122.304,395.141,-89.783,-176.757,11.396,149.480
C06320=1122.300,395.388,-89.822,-176.755,11.398,149.480
C06321=1122.296,395.635,-89.859,-176.754,11.401,149.481
C06322=1122.292,395.882,-89.898,-176.752,11.404,149.481
C06323=1122.289,396.130,-89.936,-176.751,11.407,149.481
C06324=1122.285,396.376,-89.973,-176.750,11.411,149.482
C06325=1122.281,396.624,-90.012,-176.748,11.413,149.482
C06326=1122.278,396.870,-90.050,-176.747,11.416,149.483
C06327=1122.274,397.117,-90.089,-176.746,11.419,149.483
C06328=1122.271,397.365,-90.127,-176.745,11.422,149.484
C06329=1122.266,397.612,-90.165,-176.743,11.426,149.484
C06330=1122.263,397.859,-90.203,-176.742,11.429,149.485
C06331=1122.260,398.105,-90.242,-176.741,11.432,149.485
C06332=1122.256,398.352,-90.280,-176.739,11.436,149.486
C06333=1122.252,398.600,-90.318,-176.739,11.439,149.487
C06334=1122.248,398.847,-90.356,-176.738,11.442,149.487
C06335=1122.245,399.093,-90.394,-176.736,11.445,149.488
C06336=1122.241,399.341,-90.433,-176.735,11.450,149.488
C06337=1122.238,399.588,-90.471,-176.734,11.453,149.489
C06338=1122.234,399.834,-90.510,-176.733,11.456,149.489
C06339=1122.230,400.082,-90.548,-176.732,11.460,149.490
C06340=1122.226,400.329,-90.586,-176.731,11.463,149.491
C06341=1122.224,400.576,-90.625,-176.729,11.467,149.491
C06342=1122.219,400.823,-90.663,-176.728,11.470,149.492
C06343=1122.216,401.070,-90.701,-176.728,11.474,149.493
C06344=1122.212,401.317,-90.740,-176.726,11.478,149.493
C06345=1122.209,401.563,-90.778,-176.725,11.481,149.494
C06346=1122.205,401.811,-90.816,-176.724,11.485,149.495
C06347=1122.202,402.058,-90.855,-176.723,11.488,149.495
C06348=1122.198,402.270,-90.888,-176.723,11.491,149.496
C06349=1122.195,402.482,-90.921,-176.722,11.495,149.497
C06350=1122.192,402.693,-90.954,-176.721,11.498,149.497
C06351=1122.188,402.906,-90.987,-176.720,11.501,149.498
C06352=1122.185,403.117,-91.020,-176.719,11.504,149.499
C06353=1122.182,403.329,-91.053,-176.719,11.508,149.499
C06354=1122.179,403.541,-91.085,-176.718,11.511,149.500
C06355=1122.177,403.754,-91.119,-176.717,11.514,149.501
C06356=1122.173,404.000,-91.158,-176.716,11.519,149.502
C06357=1122.169,404.248,-91.197,-176.715,11.522,149.502
C06358=1122.166,404.494,-91.235,-176.714,11.526,149.503
C06359=1122.162,404.742,-91.274,-176.713,11.531,149.504
C06360=1122.158,404.988,-91.312,-176.713,11.534,149.505
C06361=1122.154,405.235,-91.351,-176.712,11.539,149.506
C06362=1122.151,405.482,-91.390,-176.711,11.543,149.507
C06363=1122.148,405.730,-91.428,-176.710,11.547,149.507
C06364=1122.143,405.976,-91.467,-176.710,11.551,149.508
C06365=1122.140,406.223,-91.505,-176.709,11.556,149.509
C06366=1122.137,406.470,-91.544,-176.708,11.559,149.510
C06367=1122.133,406.718,-91.582,-176.707,11.564,149.511
C06368=1122.130,406.964,-91.621,-176.706,11.568,149.512
C06369=1122.126,407.210,-91.660,-176.706,11.572,149.513
C06370=1122.122,407.458,-91.698,-176.706,11.577,149.514
C06371=1122.119,407.705,-91.737,-176.705,11.581,149.515
C06372=1122.115,407.952,-91.776,-176.704,11.586,149.516
C06373=1122.111,408.199,-91.815,-176.703,11.590,149.517
C06374=1122.108,408.446,-91.854,-176.703,11.594,149.518
C06375=1122.104,408.693,-91.892,-176.702,11.599,149.519
C06376=1122.100,408.940,-91.931,-176.702,11.603,149.520
C06377=1122.097,409.186,-91.970,-176.701,11.608,149.521
C06378=1122.093,409.434,-92.008,-176.700,11.613,149.522
C06379=1122.090,409.681,-92.047,-176.700,11.618,149.523
C06380=1122.086,409.927,-92.086,-176.700,11.622,149.524
C06381=1122.082,410.174,-92.124,-176.699,11.627,149.526
C06382=1122.079,410.421,-92.163,-176.699,11.631,149.527
C06383=1122.075,410.668,-92.203,-176.698,11.636,149.528
C06384=1122.071,410.915,-92.242,-176.698,11.641,149.529
C06385=1122.068,411.163,-92.280,-176.698,11.646,149.530
C06386=1122.065,411.410,-92.319,-176.697,11.651,149.531
C06387=1122.060,411.656,-92.358,-176.696,11.656,149.532
C06388=1122.057,411.903,-92.397,-176.696,11.661,149.534
C06389=1122.054,412.149,-92.436,-176.696,11.666,149.535
C06390=1122.050,412.397,-92.474,-176.695,11.670,149.536
C06391=1122.046,412.644,-92.514,-176.695,11.676,149.537
C06392=1122.043,412.891,-92.553,-176.695,11.681,149.539
C06393=1122.040,413.138,-92.592,-176.695,11.686,149.540
C06394=1122.036,413.385,-92.631,-176.694,11.692,149.541
C06395=1122.032,413.631,-92.670,-176.694,11.697,149.542
C06396=1122.028,413.878,-92.708,-176.694,11.702,149.544
C06397=1122.026,414.126,-92.747,-176.694,11.707,149.545
C06398=1122.023,414.372,-92.787,-176.693,11.712,149.546
C06399=1122.022,414.619,-92.825,-176.694,11.717,149.548
C06400=1122.020,414.866,-92.864,-176.693,11.723,149.549
C06401=1122.020,415.113,-92.903,-176.693,11.729,149.551
C06402=1122.019,415.360,-92.941,-176.693,11.734,149.552
C06403=1122.020,415.607,-92.980,-176.693,11.739,149.553
C06404=1122.021,415.819,-93.013,-176.693,11.744,149.555
C06405=1122.022,416.031,-93.046,-176.693,11.749,149.556
C06406=1122.023,416.242,-93.078,-176.693,11.753,149.557
C06407=1122.025,416.454,-93.111,-176.693,11.758,149.558
C06408=1122.028,416.666,-93.143,-176.693,11.763,149.559
C06409=1122.031,416.878,-93.177,-176.694,11.767,149.561
C06410=1122.034,417.090,-93.209,-176.693,11.773,149.562
C06411=1122.037,417.301,-93.242,-176.693,11.778,149.563
C06412=1121.618,417.301,-93.304,-176.686,11.782,149.563
C06413=1121.614,417.089,-93.272,-176.686,11.777,149.561
C06414=1121.612,416.878,-93.240,-176.686,11.772,149.560
C06415=1121.609,416.665,-93.207,-176.686,11.767,149.559
C06416=1121.606,416.454,-93.174,-176.686,11.762,149.558
C06417=1121.604,416.242,-93.141,-176.686,11.758,149.556
C06418=1121.602,416.030,-93.108,-176.686,11.753,149.555
C06419=1121.602,415.818,-93.075,-176.686,11.748,149.554
C06420=1121.601,415.607,-93.042,-176.686,11.744,149.553
C06421=1121.600,415.360,-93.004,-176.686,11.738,149.551
C06422=1121.600,415.114,-92.965,-176.686,11.732,149.550
C06423=1121.601,414.866,-92.926,-176.686,11.727,149.549
C06424=1121.603,414.619,-92.888,-176.686,11.722,149.547
C06425=1121.604,414.372,-92.849,-176.687,11.716,149.546
C06426=1121.606,414.125,-92.810,-176.687,11.711,149.544
C06427=1121.609,413.878,-92.771,-176.687,11.706,149.543
C06428=1121.613,413.631,-92.732,-176.688,11.701,149.542
C06429=1121.616,413.384,-92.693,-176.688,11.695,149.541
C06430=1121.620,413.138,-92.653,-176.688,11.690,149.539
C06431=1121.623,412.890,-92.615,-176.689,11.685,149.538
C06432=1121.627,412.643,-92.576,-176.689,11.679,149.537
C06433=1121.630,412.396,-92.537,-176.689,11.674,149.535
C06434=1121.635,412.150,-92.498,-176.690,11.670,149.534
C06435=1121.638,411.903,-92.459,-176.690,11.664,149.533
C06436=1121.641,411.656,-92.420,-176.690,11.660,149.532
C06437=1121.645,411.409,-92.382,-176.691,11.655,149.531
C06438=1121.649,411.162,-92.342,-176.691,11.650,149.530
C06439=1121.652,410.915,-92.303,-176.692,11.645,149.528
C06440=1121.655,410.668,-92.264,-176.692,11.640,149.527
C06441=1121.660,410.421,-92.226,-176.693,11.635,149.526
C06442=1121.663,410.174,-92.187,-176.693,11.630,149.525
C06443=1121.667,409.927,-92.148,-176.694,11.626,149.524
C06444=1121.670,409.681,-92.109,-176.694,11.621,149.523
C06445=1121.674,409.433,-92.070,-176.695,11.616,149.522
C06446=1121.677,409.186,-92.031,-176.695,11.611,149.521
C06447=1121.681,408.939,-91.992,-176.696,11.607,149.520
C06448=1121.685,408.693,-91.954,-176.697,11.602,149.518
C06449=1121.688,408.446,-91.915,-176.697,11.597,149.517
C06450=1121.692,408.199,-91.876,-176.698,11.593,149.516
C06451=1121.695,407.952,-91.837,-176.698,11.589,149.515
C06452=1121.699,407.705,-91.799,-176.699,11.584,149.514
C06453=1121.702,407.458,-91.759,-176.700,11.580,149.514
C06454=1121.706,407.211,-91.722,-176.701,11.575,149.512
C06455=1121.710,406.964,-91.683,-176.702,11.571,149.512
C06456=1121.714,406.717,-91.643,-176.703,11.566,149.511
C06457=1121.717,406.470,-91.605,-176.703,11.563,149.510
C06458=1121.720,406.223,-91.566,-176.704,11.558,149.509
C06459=1121.725,405.976,-91.528,-176.705,11.554,149.508
C06460=1121.728,405.729,-91.489,-176.706,11.549,149.507
C06461=1121.731,405.482,-91.450,-176.706,11.546,149.506
C06462=1121.735,405.235,-91.412,-176.707,11.541,149.505
C06463=1121.739,404.989,-91.373,-176.708,11.537,149.504
C06464=1121.743,404.741,-91.335,-176.709,11.533,149.504
C06465=1121.746,404.495,-91.296,-176.710,11.529,149.503
C06466=1121.749,404.247,-91.258,-176.711,11.525,149.502
C06467=1121.753,404.000,-91.218,-176.711,11.521,149.501
C06468=1121.757,403.754,-91.181,-176.713,11.517,149.500
C06469=1121.760,403.542,-91.147,-176.713,11.514,149.500
C06470=1121.763,403.330,-91.114,-176.714,11.510,149.499
C06471=1121.766,403.117,-91.081,-176.715,11.507,149.498
C06472=1121.769,402.905,-91.048,-176.716,11.504,149.498
C06473=1121.772,402.694,-91.015,-176.717,11.501,149.497
C06474=1121.775,402.482,-90.983,-176.717,11.497,149.496
C06475=1121.778,402.270,-90.949,-176.718,11.494,149.496
C06476=1121.782,402.058,-90.916,-176.719,11.491,149.495
C06477=1121.785,401.811,-90.877,-176.720,11.487,149.494
C06478=1121.789,401.565,-90.839,-176.721,11.484,149.494
C06479=1121.793,401.317,-90.801,-176.722,11.479,149.493
C06480=1121.796,401.070,-90.763,-176.723,11.476,149.492
C06481=1121.800,400.823,-90.723,-176.725,11.472,149.492
C06482=1121.803,400.576,-90.686,-176.725,11.469,149.491
C06483=1121.807,400.329,-90.647,-176.727,11.465,149.490
C06484=1121.810,400.082,-90.609,-176.728,11.462,149.490
C06485=1121.815,399.835,-90.571,-176.730,11.458,149.489
C06486=1121.818,399.588,-90.533,-176.730,11.455,149.489
C06487=1121.822,399.341,-90.493,-176.731,11.452,149.488
C06488=1121.825,399.094,-90.456,-176.733,11.448,149.487
C06489=1121.829,398.847,-90.417,-176.734,11.445,149.487
C06490=1121.832,398.600,-90.379,-176.735,11.442,149.486
C06491=1121.837,398.353,-90.340,-176.737,11.438,149.486
C06492=1121.840,398.106,-90.302,-176.738,11.435,149.485
C06493=1121.844,397.858,-90.264,-176.739,11.432,149.485
C06494=1121.847,397.612,-90.226,-176.741,11.428,149.484
C06495=1121.851,397.365,-90.187,-176.742,11.425,149.484
C06496=1121.854,397.118,-90.149,-176.743,11.422,149.483
C06497=1121.858,396.871,-90.112,-176.744,11.418,149.483
C06498=1121.862,396.623,-90.073,-176.746,11.415,149.482
C06499=1121.865,396.377,-90.034,-176.747,11.412,149.482
C06500=1121.870,396.130,-89.996,-176.748,11.409,149.481
C06501=1121.873,395.883,-89.958,-176.750,11.406,149.481
C06502=1121.877,395.635,-89.920,-176.751,11.403,149.480
C06503=1121.880,395.389,-89.882,-176.752,11.400,149.480
C06504=1121.884,395.141,-89.844,-176.753,11.397,149.479
C06505=1121.888,394.895,-89.805,-176.756,11.393,149.479
C06506=1121.891,394.648,-89.767,-176.757,11.390,149.478
C06507=1121.895,394.400,-89.729,-176.758,11.388,149.478
C06508=1121.899,394.154,-89.691,-176.760,11.385,149.478
C06509=1121.902,393.906,-89.653,-176.761,11.382,149.477
C06510=1121.906,393.659,-89.615,-176.762,11.379,149.477
C06511=1121.910,393.412,-89.577,-176.764,11.377,149.477
C06512=1121.913,393.165,-89.539,-176.766,11.373,149.476
C06513=1121.917,392.918,-89.501,-176.767,11.371,149.476
C06514=1121.921,392.671,-89.463,-176.769,11.368,149.476
C06515=1121.924,392.424,-89.426,-176.770,11.365,149.475
C06516=1121.928,392.177,-89.387,-176.772,11.362,149.475
C06517=1121.931,391.929,-89.349,-176.773,11.360,149.475
C06518=1121.935,391.683,-89.312,-176.775,11.357,149.474
C06519=1121.939,391.435,-89.273,-176.777,11.355,149.474
C06520=1121.943,391.189,-89.235,-176.778,11.352,149.474
C06521=1121.946,390.941,-89.198,-176.780,11.349,149.474
C06522=1121.950,390.694,-89.159,-176.781,11.347,149.473
C06523=1121.954,390.447,-89.121,-176.783,11.344,149.473
C06524=1121.957,390.200,-89.084,-176.784,11.342,149.473
C06525=1121.961,389.988,-89.051,-176.786,11.339,149.473
C06526=1121.963,389.776,-89.018,-176.787,11.338,149.473
C06527=1121.966,389.564,-88.986,-176.789,11.335,149.472
C06528=1121.970,389.351,-88.953,-176.791,11.333,149.472
C06529=1121.973,389.140,-88.921,-176.792,11.331,149.472
C06530=1121.977,388.928,-88.889,-176.794,11.328,149.472
C06531=1121.979,388.716,-88.856,-176.795,11.327,149.472
C06532=1121.983,388.504,-88.824,-176.797,11.324,149.471
C06533=1121.986,388.257,-88.786,-176.799,11.322,149.471
C06534=1121.990,388.010,-88.749,-176.800,11.319,149.471
C06535=1121.994,387.762,-88.710,-176.802,11.317,149.471
C06536=1121.998,387.515,-88.673,-176.803,11.315,149.471
C06537=1122.001,387.268,-88.635,-176.805,11.313,149.471
C06538=1122.005,387.022,-88.597,-176.807,11.311,149.471
C06539=1122.008,386.774,-88.559,-176.809,11.308,149.470
C06540=1122.013,386.527,-88.522,-176.811,11.306,149.470
C06541=1122.016,386.280,-88.484,-176.813,11.304,149.470
C06542=1122.020,386.033,-88.446,-176.815,11.302,149.470
C06543=1122.023,385.786,-88.408,-176.817,11.299,149.470
C06544=1122.027,385.539,-88.371,-176.819,11.297,149.470
C06545=1122.030,385.291,-88.333,-176.820,11.295,149.470
C06546=1122.035,385.044,-88.295,-176.822,11.293,149.470
C06547=1122.038,384.797,-88.257,-176.824,11.291,149.470
C06548=1122.042,384.550,-88.221,-176.826,11.289,149.470
C06549=1122.045,384.303,-88.183,-176.828,11.287,149.470
C06550=1122.049,384.056,-88.145,-176.830,11.284,149.470
C06551=1122.052,383.809,-88.107,-176.832,11.283,149.470
C06552=1122.056,383.562,-88.070,-176.834,11.281,149.470
C06553=1122.060,383.314,-88.032,-176.836,11.279,149.470
C06554=1122.064,383.067,-87.994,-176.839,11.276,149.470
C06555=1122.067,382.820,-87.957,-176.842,11.273,149.470
C06556=1122.071,382.573,-87.919,-176.845,11.270,149.470
C06557=1122.075,382.326,-87.882,-176.848,11.269,149.470
C06558=1122.078,382.079,-87.844,-176.850,11.266,149.470
C06559=1122.082,381.832,-87.807,-176.853,11.263,149.470
C06560=1122.086,381.584,-87.770,-176.857,11.261,149.470
C06561=1122.089,381.337,-87.732,-176.860,11.258,149.470
C06562=1122.093,381.090,-87.695,-176.862,11.256,149.470
C06563=1122.097,380.843,-87.657,-176.865,11.253,149.470
C06564=1122.101,380.596,-87.620,-176.868,11.251,149.471
C06565=1122.104,380.349,-87.583,-176.871,11.248,149.471
C06566=1122.108,380.101,-87.546,-176.875,11.246,149.471
C06567=1122.112,379.855,-87.508,-176.877,11.244,149.471
C06568=1122.115,379.607,-87.471,-176.880,11.241,149.471
C06569=1122.119,379.360,-87.433,-176.883,11.238,149.471
C06570=1122.123,379.112,-87.396,-176.886,11.236,149.471
C06571=1122.126,378.866,-87.358,-176.889,11.233,149.471
C06572=1122.131,378.619,-87.322,-176.892,11.231,149.472
C06573=1122.134,378.371,-87.284,-176.895,11.229,149.472
C06574=1122.138,378.124,-87.247,-176.898,11.226,149.472
C06575=1122.142,377.877,-87.210,-176.901,11.223,149.472
C06576=1122.145,377.629,-87.173,-176.904,11.222,149.472
C06577=1122.149,377.383,-87.135,-176.907,11.219,149.472
C06578=1122.153,377.135,-87.098,-176.910,11.216,149.472
C06579=1122.157,376.887,-87.061,-176.914,11.214,149.473
C06580=1122.161,376.641,-87.024,-176.917,11.211,149.473
C06581=1122.164,376.428,-86.992,-176.919,11.209,149.473
C06582=1122.168,376.217,-86.960,-176.922,11.208,149.473
C06583=1122.170,376.005,-86.928,-176.924,11.206,149.473
C06584=1122.174,375.792,-86.897,-176.927,11.203,149.473
C06585=1122.176,375.580,-86.865,-176.930,11.201,149.474
C06586=1122.180,375.367,-86.833,-176.932,11.200,149.474
C06587=1122.183,375.156,-86.801,-176.935,11.197,149.474
C06588=1122.186,374.944,-86.769,-176.938,11.195,149.474
C06589=1122.190,374.696,-86.732,-176.941,11.193,149.474
C06590=1122.194,374.449,-86.695,-176.943,11.190,149.474
C06591=1122.198,374.201,-86.658,-176.947,11.188,149.474
C06592=1122.202,373.954,-86.621,-176.950,11.186,149.475
C06593=1122.205,373.707,-86.585,-176.953,11.183,149.475
C06594=1122.209,373.459,-86.548,-176.957,11.181,149.475
C06595=1122.213,373.213,-86.510,-176.960,11.178,149.475
C06596=1122.217,372.966,-86.474,-176.963,11.176,149.476
C06597=1122.221,372.718,-86.437,-176.966,11.174,149.476
C06598=1122.223,372.471,-86.400,-176.969,11.171,149.476
C06599=1122.228,372.224,-86.363,-176.972,11.169,149.476
C06600=1122.232,371.976,-86.326,-176.976,11.166,149.476
C06601=1122.235,371.730,-86.290,-176.979,11.164,149.477
C06602=1122.239,371.482,-86.253,-176.982,11.162,149.477
C06603=1122.243,371.235,-86.216,-176.985,11.160,149.477
C06604=1122.247,370.987,-86.179,-176.988,11.157,149.477
C06605=1122.250,370.740,-86.143,-176.992,11.155,149.477
C06606=1122.254,370.493,-86.106,-176.995,11.152,149.478
C06607=1122.258,370.246,-86.069,-176.998,11.150,149.478
C06608=1122.261,369.998,-86.033,-177.002,11.147,149.478
C06609=1122.265,369.751,-85.996,-177.004,11.146,149.478
C06610=1122.270,369.503,-85.960,-177.008,11.143,149.479
C06611=1122.273,369.257,-85.923,-177.011,11.141,149.479
C06612=1122.277,369.009,-85.886,-177.014,11.138,149.479
C06613=1122.281,368.762,-85.850,-177.017,11.136,149.479
C06614=1122.284,368.515,-85.813,-177.021,11.133,149.479
C06615=1122.288,368.267,-85.776,-177.024,11.131,149.480
C06616=1122.292,368.020,-85.741,-177.027,11.128,149.480
C06617=1122.296,367.773,-85.704,-177.030,11.127,149.480
C06618=1122.300,367.526,-85.667,-177.033,11.124,149.480
C06619=1122.303,367.279,-85.631,-177.037,11.122,149.480
C06620=1122.308,367.031,-85.594,-177.040,11.120,149.481
C06621=1122.311,366.784,-85.558,-177.044,11.117,149.481
C06622=1122.314,366.536,-85.521,-177.047,11.115,149.481
C06623=1122.318,366.289,-85.485,-177.050,11.112,149.481
C06624=1122.322,366.041,-85.449,-177.054,11.110,149.482
C06625=1122.326,365.794,-85.412,-177.057,11.107,149.482
C06626=1122.330,365.547,-85.375,-177.060,11.105,149.482
C06627=1122.334,365.300,-85.339,-177.063,11.103,149.483
C06628=1122.337,365.053,-85.303,-177.066,11.101,149.483
C06629=1122.342,364.805,-85.267,-177.070,11.098,149.483
C06630=1122.345,364.558,-85.231,-177.073,11.096,149.483
C06631=1122.349,364.311,-85.194,-177.076,11.094,149.483
C06632=1122.353,364.063,-85.158,-177.080,11.091,149.484
C06633=1122.356,363.816,-85.122,-177.083,11.089,149.484
C06634=1122.361,363.569,-85.086,-177.087,11.086,149.484
C06635=1122.364,363.322,-85.050,-177.090,11.084,149.484
C06636=1122.368,363.073,-85.013,-177.093,11.081,149.485
C06637=1122.371,362.861,-84.982,-177.096,11.080,149.485
C06638=1122.374,362.649,-84.951,-177.099,11.077,149.485
C06639=1122.377,362.437,-84.920,-177.102,11.076,149.485
C06640=1122.380,362.224,-84.889,-177.105,11.073,149.486
C06641=1122.384,362.012,-84.858,-177.108,11.071,149.486
C06642=1122.387,361.800,-84.827,-177.111,11.070,149.486
C06643=1122.391,361.588,-84.796,-177.114,11.067,149.486
C06644=1122.394,361.375,-84.765,-177.116,11.065,149.486
C06645=1122.397,361.128,-84.729,-177.120,11.063,149.487
C06646=1122.401,360.880,-84.694,-177.123,11.061,149.487
C06647=1122.405,360.633,-84.657,-177.127,11.058,149.487
C06648=1122.409,360.385,-84.621,-177.130,11.056,149.487
C06649=1122.413,360.138,-84.586,-177.134,11.054,149.488
C06650=1122.417,359.891,-84.549,-177.137,11.051,149.488
C06651=1122.420,359.643,-84.513,-177.140,11.049,149.488
C06652=1122.424,359.396,-84.478,-177.143,11.046,149.488
C06653=1122.428,359.149,-84.441,-177.147,11.044,149.489
C06654=1122.432,358.901,-84.405,-177.150,11.042,149.489
C06655=1122.435,358.654,-84.370,-177.154,11.039,149.489
C06656=1122.439,358.406,-84.334,-177.157,11.037,149.490
C06657=1122.444,358.160,-84.298,-177.161,11.033,149.490
C06658=1122.447,357.912,-84.262,-177.165,11.031,149.490
C06659=1122.451,357.665,-84.227,-177.168,11.029,149.490
C06660=1122.455,357.417,-84.191,-177.171,11.026,149.491
C06661=1122.458,357.170,-84.156,-177.175,11.024,149.491
C06662=1122.463,356.922,-84.120,-177.178,11.022,149.491
C06663=1122.466,356.674,-84.084,-177.182,11.019,149.491
C06664=1122.470,356.427,-84.048,-177.185,11.017,149.492
C06665=1122.473,356.180,-84.012,-177.188,11.014,149.492
C06666=1122.478,355.933,-83.977,-177.192,11.012,149.492
C06667=1122.482,355.685,-83.941,-177.195,11.010,149.492
C06668=1122.486,355.438,-83.905,-177.199,11.007,149.493
C06669=1122.489,355.190,-83.870,-177.203,11.004,149.493
C06670=1122.493,354.943,-83.834,-177.206,11.002,149.493
C06671=1122.497,354.695,-83.799,-177.210,10.999,149.494
C06672=1122.500,354.448,-83.763,-177.213,10.997,149.494
C06673=1122.505,354.201,-83.728,-177.216,10.995,149.494
C06674=1122.508,353.953,-83.692,-177.219,10.992,149.494
C06675=1122.512,353.706,-83.657,-177.223,10.990,149.494
C06676=1122.516,353.458,-83.621,-177.227,10.987,149.495
C06677=1122.520,353.211,-83.585,-177.230,10.984,149.495
C06678=1122.525,352.963,-83.551,-177.234,10.982,149.495
C06679=1122.528,352.716,-83.515,-177.237,10.979,149.495
C06680=1122.532,352.468,-83.480,-177.240,10.977,149.496
C06681=1122.536,352.221,-83.444,-177.245,10.974,149.496
C06682=1122.539,351.973,-83.408,-177.248,10.971,149.496
C06683=1122.544,351.726,-83.373,-177.251,10.969,149.496
C06684=1122.548,351.478,-83.338,-177.255,10.967,149.497
C06685=1122.551,351.231,-83.303,-177.258,10.964,149.497
C06686=1122.555,350.983,-83.267,-177.262,10.961,149.497
C06687=1122.559,350.736,-83.232,-177.266,10.959,149.498
C06688=1122.563,350.488,-83.197,-177.269,10.956,149.498
C06689=1122.567,350.241,-83.162,-177.272,10.954,149.498
C06690=1122.570,349.993,-83.126,-177.276,10.951,149.498
C06691=1122.575,349.747,-83.091,-177.279,10.948,149.498
C06692=1122.578,349.499,-83.057,-177.283,10.946,149.499
C06693=1122.582,349.286,-83.027,-177.286,10.943,149.499
C06694=1122.585,349.074,-82.995,-177.288,10.941,149.499
C06695=1122.588,348.861,-82.966,-177.291,10.939,149.499
C06696=1122.592,348.649,-82.936,-177.294,10.937,149.499
C06697=1122.595,348.436,-82.906,-177.297,10.935,149.500
C06698=1122.599,348.223,-82.875,-177.299,10.933,149.500
C06699=1122.602,348.011,-82.846,-177.302,10.931,149.500
C06700=1122.605,347.799,-82.815,-177.305,10.929,149.500
C06701=1122.609,347.551,-82.781,-177.308,10.926,149.500
C06702=1122.612,347.304,-82.745,-177.312,10.924,149.501
C06703=1122.617,347.056,-82.711,-177.315,10.921,149.501
C06704=1122.621,346.809,-82.675,-177.318,10.919,149.501
C06705=1122.625,346.561,-82.640,-177.321,10.916,149.501
C06706=1122.629,346.314,-82.605,-177.324,10.914,149.501
C06707=1122.632,346.066,-82.571,-177.328,10.911,149.502
C06708=1122.636,345.819,-82.535,-177.331,10.909,149.502
C06709=1122.640,345.571,-82.501,-177.334,10.906,149.502
C06710=1122.644,345.323,-82.466,-177.338,10.904,149.502
C06711=1122.649,345.076,-82.431,-177.341,10.901,149.502
C06712=1122.652,344.828,-82.397,-177.344,10.899,149.502
C06713=1122.655,344.581,-82.361,-177.347,10.897,149.503
C06714=1122.660,344.333,-82.327,-177.350,10.895,149.503
C06715=1122.664,344.085,-82.292,-177.353,10.892,149.503
C06716=1122.668,343.839,-82.257,-177.356,10.890,149.503
C06717=1122.671,343.591,-82.222,-177.359,10.887,149.503
C06718=1122.675,343.343,-82.187,-177.363,10.884,149.504
C06719=1122.679,343.096,-82.153,-177.366,10.882,149.504
C06720=1122.683,342.848,-82.118,-177.369,10.879,149.504
C06721=1122.688,342.601,-82.084,-177.373,10.877,149.504
C06722=1122.691,342.352,-82.049,-177.376,10.874,149.504
C06723=1122.695,342.106,-82.014,-177.379,10.872,149.505
C06724=1122.699,341.858,-81.979,-177.382,10.869,149.505
C06725=1122.704,341.610,-81.945,-177.386,10.867,149.505
C06726=1122.707,341.363,-81.911,-177.389,10.864,149.505
C06727=1122.711,341.115,-81.876,-177.392,10.862,149.505
C06728=1122.715,340.867,-81.841,-177.395,10.859,149.506
C06729=1122.719,340.621,-81.807,-177.398,10.857,149.506
C06730=1122.723,340.372,-81.772,-177.401,10.855,149.506
C06731=1122.727,340.125,-81.738,-177.404,10.853,149.506
C06732=1122.731,339.877,-81.703,-177.407,10.850,149.506
C06733=1122.735,339.630,-81.669,-177.411,10.847,149.507
C06734=1122.738,339.382,-81.635,-177.414,10.845,149.507
C06735=1122.743,339.135,-81.600,-177.417,10.842,149.507
C06736=1122.746,338.887,-81.566,-177.421,10.840,149.507
C06737=1122.751,338.639,-81.531,-177.423,10.837,149.507
C06738=1122.755,338.391,-81.497,-177.427,10.835,149.508
C06739=1122.759,338.144,-81.463,-177.430,10.832,149.508
C06740=1122.763,337.896,-81.428,-177.433,10.830,149.508
C06741=1122.766,337.649,-81.394,-177.436,10.827,149.508
C06742=1122.770,337.401,-81.359,-177.440,10.825,149.508
C06743=1122.774,337.154,-81.325,-177.443,10.822,149.509
C06744=1122.779,336.906,-81.291,-177.446,10.820,149.509
C06745=1122.782,336.658,-81.257,-177.450,10.817,149.509
C06746=1122.786,336.411,-81.223,-177.452,10.815,149.509
C06747=1122.790,336.163,-81.188,-177.455,10.813,149.509
C06748=1122.794,335.916,-81.154,-177.459,10.810,149.510
C06749=1122.798,335.635,-81.115,-177.463,10.807,149.510
C06750=1122.803,335.354,-81.076,-177.466,10.805,149.510
C06751=1122.807,335.069,-81.037,-177.470,10.801,149.510
C06752=1122.812,334.784,-80.998,-177.473,10.799,149.511
C06753=1122.816,334.500,-80.959,-177.477,10.796,149.511
C06754=1122.821,334.215,-80.919,-177.480,10.793,149.511
C06755=1122.825,333.967,-80.886,-177.484,10.791,149.511
C06756=1122.829,333.719,-80.851,-177.487,10.788,149.511
C06757=1122.833,333.472,-80.817,-177.490,10.786,149.512
C06758=1122.836,333.224,-80.783,-177.493,10.783,149.512
C06759=1122.841,332.976,-80.749,-177.497,10.781,149.512
C06760=1122.845,332.729,-80.715,-177.499,10.778,149.512
C06761=1122.848,332.482,-80.681,-177.503,10.775,149.512
C06762=1122.853,332.233,-80.647,-177.506,10.773,149.513
C06763=1122.857,331.986,-80.613,-177.509,10.770,149.513
C06764=1122.860,331.739,-80.580,-177.512,10.768,149.513
C06765=1122.865,331.490,-80.545,-177.516,10.765,149.513
C06766=1122.868,331.243,-80.512,-177.519,10.763,149.513
C06767=1122.873,330.995,-80.478,-177.522,10.760,149.513
C06768=1122.876,330.747,-80.444,-177.525,10.758,149.514
C06769=1122.881,330.499,-80.410,-177.528,10.756,149.514
C06770=1122.885,330.252,-80.377,-177.531,10.754,149.514
C06771=1122.888,330.005,-80.343,-177.534,10.751,149.514
C06772=1122.892,329.756,-80.309,-177.537,10.748,149.515
C06773=1122.896,329.509,-80.275,-177.541,10.746,149.515
C06774=1122.901,329.261,-80.242,-177.544,10.743,149.515
C06775=1122.904,329.014,-80.207,-177.547,10.741,149.515
C06776=1122.908,328.766,-80.174,-177.550,10.738,149.515
C06777=1122.912,328.518,-80.141,-177.553,10.735,149.515
C06778=1122.917,328.271,-80.107,-177.557,10.733,149.516
C06779=1122.920,328.022,-80.073,-177.560,10.731,149.516
C06780=1122.924,327.775,-80.039,-177.563,10.728,149.516
C06781=1122.928,327.527,-80.006,-177.566,10.725,149.516
C06782=1122.932,327.280,-79.973,-177.570,10.723,149.516
C06783=1122.936,327.033,-79.939,-177.573,10.720,149.517
C06784=1122.940,326.784,-79.905,-177.576,10.718,149.517
C06785=1122.945,326.536,-79.872,-177.578,10.716,149.517
C06786=1122.948,326.289,-79.838,-177.582,10.714,149.517
C06787=1122.953,326.041,-79.805,-177.585,10.711,149.517
C06788=1122.957,325.793,-79.772,-177.588,10.708,149.518
C06789=1122.960,325.546,-79.737,-177.591,10.706,149.518
C06790=1122.964,325.298,-79.704,-177.594,10.703,149.518
C06791=1122.968,325.050,-79.671,-177.598,10.701,149.518
C06792=1122.972,324.802,-79.638,-177.601,10.698,149.518
C06793=1122.976,324.555,-79.604,-177.604,10.695,149.518
C06794=1122.980,324.307,-79.570,-177.607,10.693,149.519
C06795=1122.984,324.059,-79.537,-177.610,10.691,149.519
C06796=1122.988,323.811,-79.504,-177.613,10.688,149.519
C06797=1122.992,323.564,-79.471,-177.617,10.685,149.519
C06798=1122.996,323.317,-79.437,-177.620,10.683,149.519
C06799=1123.000,323.069,-79.404,-177.623,10.680,149.520
C06800=1123.004,322.821,-79.371,-177.626,10.678,149.520
C06801=1123.008,322.573,-79.337,-177.629,10.676,149.520
C06802=1123.012,322.325,-79.304,-177.632,10.673,149.520
C06803=1123.015,322.112,-79.275,-177.635,10.671,149.520
C06804=1123.019,321.900,-79.247,-177.638,10.669,149.520
C06805=1123.023,321.687,-79.219,-177.640,10.667,149.521
C06806=1123.026,321.474,-79.190,-177.643,10.664,149.521
C06807=1123.029,321.261,-79.162,-177.645,10.662,149.521
C06808=1123.032,321.048,-79.133,-177.649,10.660,149.521
C06809=1123.036,320.836,-79.104,-177.651,10.658,149.521
C06810=1123.039,320.622,-79.077,-177.654,10.656,149.522
C06811=1123.043,320.375,-79.043,-177.657,10.653,149.522
C06812=1123.047,320.127,-79.010,-177.660,10.651,149.522
C06813=1123.051,319.879,-78.977,-177.663,10.649,149.522
C06814=1123.056,319.631,-78.944,-177.666,10.646,149.522
C06815=1123.060,319.384,-78.911,-177.670,10.643,149.522
C06816=1123.064,319.136,-78.878,-177.673,10.641,149.522
C06817=1123.067,318.889,-78.845,-177.676,10.638,149.523
C06818=1123.071,318.641,-78.812,-177.679,10.636,149.523
C06819=1123.076,318.393,-78.779,-177.682,10.633,149.523
C06820=1123.080,318.145,-78.746,-177.685,10.630,149.523
C06821=1123.084,317.897,-78.713,-177.689,10.628,149.524
C06822=1123.088,317.650,-78.681,-177.691,10.626,149.524
C06823=1123.092,317.402,-78.648,-177.694,10.624,149.524
C06824=1123.096,317.154,-78.614,-177.697,10.621,149.524
C06825=1123.100,316.906,-78.581,-177.701,10.618,149.524
C06826=1123.104,316.658,-78.549,-177.704,10.616,149.524
C06827=1123.108,316.411,-78.516,-177.707,10.613,149.525
C06828=1123.112,316.163,-78.483,-177.710,10.611,149.525
C06829=1123.116,315.915,-78.450,-177.713,10.608,149.525
C06830=1123.120,315.667,-78.418,-177.716,10.605,149.525
C06831=1123.124,315.419,-78.385,-177.720,10.603,149.525
C06832=1123.128,315.172,-78.352,-177.723,10.600,149.525
C06833=1123.132,314.924,-78.320,-177.726,10.598,149.526
C06834=1123.136,314.676,-78.287,-177.729,10.595,149.526
C06835=1123.140,314.428,-78.254,-177.732,10.593,149.526
C06836=1123.144,314.180,-78.222,-177.735,10.591,149.526
C06837=1123.148,313.932,-78.189,-177.738,10.588,149.526
C06838=1123.152,313.684,-78.156,-177.741,10.586,149.527
C06839=1123.156,313.437,-78.124,-177.744,10.583,149.527
C06840=1123.160,313.189,-78.090,-177.747,10.581,149.527
C06841=1123.164,312.941,-78.058,-177.751,10.578,149.527
C06842=1123.168,312.693,-78.025,-177.754,10.575,149.527
C06843=1123.172,312.445,-77.993,-177.757,10.573,149.528
C06844=1123.176,312.198,-77.961,-177.760,10.570,149.528
C06845=1123.181,311.950,-77.928,-177.763,10.568,149.528
C06846=1123.185,311.702,-77.895,-177.767,10.565,149.528
C06847=1123.188,311.454,-77.863,-177.770,10.562,149.528
C06848=1123.193,311.206,-77.830,-177.773,10.560,149.528
C06849=1123.196,310.958,-77.798,-177.775,10.558,149.529
C06850=1123.201,310.710,-77.766,-177.779,10.556,149.529
C06851=1123.204,310.462,-77.733,-177.781,10.553,149.529
C06852=1123.209,310.214,-77.701,-177.785,10.550,149.529
C06853=1123.213,309.967,-77.668,-177.788,10.548,149.529
C06854=1123.217,309.719,-77.636,-177.791,10.545,149.529
C06855=1123.221,309.471,-77.604,-177.794,10.543,149.530
C06856=1123.225,309.223,-77.571,-177.797,10.540,149.530
C06857=1123.229,308.975,-77.539,-177.801,10.538,149.530
C06858=1123.233,308.727,-77.507,-177.804,10.535,149.530
C06859=1123.237,308.514,-77.480,-177.806,10.533,149.530
C06860=1123.240,308.302,-77.451,-177.809,10.530,149.531
C06861=1123.244,308.089,-77.424,-177.812,10.528,149.531
C06862=1123.247,307.876,-77.396,-177.814,10.527,149.531
C06863=1123.251,307.662,-77.368,-177.817,10.524,149.531
C06864=1123.255,307.450,-77.341,-177.819,10.522,149.531
C06865=1123.258,307.237,-77.313,-177.822,10.520,149.531
C06866=1123.261,307.024,-77.286,-177.825,10.517,149.531
C06867=1123.266,306.776,-77.254,-177.828,10.515,149.532
C06868=1123.269,306.528,-77.221,-177.831,10.512,149.532
C06869=1123.274,306.280,-77.189,-177.835,10.510,149.532
C06870=1123.277,306.032,-77.157,-177.837,10.508,149.532
C06871=1123.282,305.785,-77.125,-177.840,10.505,149.532
C06872=1123.286,305.536,-77.093,-177.843,10.503,149.533
C06873=1123.290,305.288,-77.061,-177.847,10.500,149.533
C06874=1123.294,305.040,-77.028,-177.849,10.497,149.533
C06875=1123.299,304.793,-76.997,-177.853,10.495,149.533
C06876=1123.302,304.545,-76.964,-177.856,10.493,149.533
C06877=1123.306,304.297,-76.932,-177.859,10.490,149.533
C06878=1123.311,304.050,-76.900,-177.862,10.487,149.534
C06879=1123.314,303.801,-76.869,-177.865,10.485,149.534
C06880=1123.318,303.553,-76.837,-177.869,10.482,149.534
C06881=1123.323,303.305,-76.804,-177.872,10.479,149.534
C06882=1123.327,303.058,-76.773,-177.874,10.478,149.534
C06883=1123.331,302.810,-76.741,-177.877,10.475,149.535
C06884=1123.335,302.561,-76.709,-177.881,10.473,149.535
C06885=1123.339,302.314,-76.677,-177.884,10.470,149.535
C06886=1123.343,302.065,-76.646,-177.887,10.467,149.535
C06887=1123.347,301.817,-76.614,-177.890,10.465,149.535
C06888=1123.352,301.570,-76.582,-177.893,10.462,149.535
C06889=1123.356,301.322,-76.550,-177.896,10.459,149.536
C06890=1123.359,301.074,-76.518,-177.899,10.457,149.536
C06891=1123.364,300.826,-76.487,-177.902,10.454,149.536
C06892=1123.368,300.578,-76.454,-177.906,10.452,149.536
C06893=1123.373,300.331,-76.423,-177.909,10.449,149.536
C06894=1123.377,300.082,-76.392,-177.911,10.447,149.537
C06895=1123.380,299.834,-76.360,-177.914,10.445,149.537
C06896=1123.385,299.587,-76.329,-177.918,10.442,149.537
C06897=1123.388,299.339,-76.297,-177.920,10.439,149.537
C06898=1123.393,299.090,-76.264,-177.924,10.437,149.537
C06899=1123.397,298.842,-76.233,-177.927,10.434,149.537
C06900=1123.401,298.594,-76.202,-177.930,10.432,149.538
C06901=1123.405,298.347,-76.170,-177.933,10.429,149.538
C06902=1123.409,298.098,-76.139,-177.936,10.427,149.538
C06903=1123.413,297.850,-76.107,-177.939,10.424,149.538
C06904=1123.417,297.603,-76.076,-177.943,10.421,149.538
C06905=1123.421,297.354,-76.045,-177.945,10.419,149.538
C06906=1123.426,297.107,-76.013,-177.948,10.417,149.539
C06907=1123.429,296.859,-75.981,-177.951,10.414,149.539
C06908=1123.434,296.611,-75.950,-177.955,10.412,149.539
C06909=1123.438,296.363,-75.919,-177.957,10.409,149.539
C06910=1123.441,296.115,-75.887,-177.961,10.407,149.539
C06911=1123.447,295.866,-75.855,-177.964,10.404,149.539
C06912=1123.450,295.618,-75.824,-177.967,10.401,149.540
C06913=1123.455,295.370,-75.793,-177.970,10.399,149.540
C06914=1123.459,295.122,-75.761,-177.973,10.396,149.540
C06915=1123.462,294.910,-75.735,-177.976,10.394,149.540
C06916=1123.465,294.696,-75.708,-177.978,10.392,149.540
C06917=1123.469,294.483,-75.681,-177.981,10.390,149.541
C06918=1123.473,294.271,-75.654,-177.984,10.388,149.541
C06919=1123.476,294.057,-75.627,-177.986,10.386,149.541
C06920=1123.480,293.844,-75.600,-177.989,10.383,149.541
C06921=1123.483,293.631,-75.573,-177.992,10.381,149.541
C06922=1123.487,293.418,-75.546,-177.994,10.379,149.541
C06923=1123.490,293.170,-75.515,-177.997,10.377,149.541
C06924=1123.495,292.922,-75.484,-178.000,10.374,149.542
C06925=1123.499,292.673,-75.453,-178.003,10.371,149.542
C06926=1123.503,292.426,-75.422,-178.006,10.369,149.542
C06927=1123.508,292.178,-75.391,-178.009,10.366,149.542
C06928=1123.512,291.930,-75.359,-178.013,10.364,149.542
C06929=1123.516,291.682,-75.328,-178.016,10.361,149.542
C06930=1123.520,291.433,-75.297,-178.019,10.359,149.543
C06931=1123.524,291.186,-75.266,-178.022,10.356,149.543
C06932=1123.528,290.938,-75.235,-178.025,10.353,149.543
C06933=1123.532,290.690,-75.204,-178.027,10.351,149.543
C06934=1123.536,290.441,-75.173,-178.031,10.349,149.544
C06935=1123.541,290.194,-75.142,-178.034,10.346,149.544
C06936=1123.545,289.945,-75.111,-178.037,10.344,149.544
C06937=1123.549,289.697,-75.081,-178.040,10.341,149.544
C06938=1123.553,289.449,-75.050,-178.043,10.338,149.544
C06939=1123.557,289.201,-75.018,-178.046,10.336,149.544
C06940=1123.561,288.953,-74.987,-178.049,10.333,149.544
C06941=1123.565,288.705,-74.956,-178.053,10.331,149.545
C06942=1123.569,288.457,-74.926,-178.056,10.328,149.545
C06943=1123.574,288.209,-74.895,-178.058,10.326,149.545
C06944=1123.578,287.961,-74.863,-178.061,10.324,149.545
C06945=1123.582,287.713,-74.833,-178.064,10.321,149.545
C06946=1123.586,287.466,-74.802,-178.067,10.318,149.546
C06947=1123.590,287.217,-74.771,-178.070,10.316,149.546
C06948=1123.595,286.969,-74.740,-178.074,10.313,149.546
C06949=1123.599,286.721,-74.710,-178.077,10.310,149.546
C06950=1123.603,286.473,-74.679,-178.080,10.308,149.546
C06951=1123.607,286.225,-74.648,-178.083,10.305,149.546
C06952=1123.611,285.977,-74.618,-178.086,10.303,149.547
C06953=1123.615,285.728,-74.587,-178.089,10.301,149.547
C06954=1123.620,285.480,-74.556,-178.091,10.298,149.547
C06955=1123.624,285.233,-74.526,-178.095,10.296,149.547
C06956=1123.628,284.984,-74.495,-178.098,10.293,149.547
C06957=1123.632,284.736,-74.464,-178.101,10.290,149.548
C06958=1123.636,284.488,-74.434,-178.104,10.288,149.548
C06959=1123.640,284.240,-74.403,-178.107,10.285,149.548
C06960=1123.644,283.992,-74.373,-178.110,10.283,149.548
C06961=1123.649,283.744,-74.342,-178.113,10.280,149.548
C06962=1123.653,283.496,-74.311,-178.117,10.277,149.548
C06963=1123.657,283.248,-74.281,-178.119,10.275,149.548
C06964=1123.661,282.999,-74.251,-178.122,10.273,149.549
C06965=1123.665,282.752,-74.221,-178.125,10.270,149.549
C06966=1123.669,282.503,-74.189,-178.129,10.268,149.549
C06967=1123.673,282.255,-74.159,-178.131,10.265,149.549
C06968=1123.678,282.007,-74.128,-178.134,10.262,149.549
C06969=1123.683,281.759,-74.098,-178.138,10.260,149.550
C06970=1123.687,281.511,-74.068,-178.141,10.257,149.550
C06971=1123.690,281.297,-74.041,-178.143,10.255,149.550
C06972=1123.693,281.085,-74.015,-178.146,10.253,149.550
C06973=1123.697,280.871,-73.989,-178.150,10.250,149.550
C06974=1123.701,280.658,-73.964,-178.152,10.248,149.551
C06975=1123.705,280.445,-73.937,-178.155,10.246,149.551
C06976=1123.708,280.231,-73.911,-178.158,10.243,149.551
C06977=1123.712,280.018,-73.885,-178.161,10.241,149.551
C06978=1123.715,279.805,-73.859,-178.164,10.238,149.551
C06979=1123.720,279.557,-73.829,-178.167,10.236,149.551
C06980=1123.724,279.309,-73.799,-178.170,10.232,149.551
C06981=1123.728,279.061,-73.769,-178.174,10.230,149.552
C06982=1123.732,278.812,-73.738,-178.177,10.227,149.552
C06983=1123.736,278.564,-73.708,-178.180,10.225,149.552
C06984=1123.741,278.316,-73.678,-178.183,10.222,149.552
C06985=1123.745,278.068,-73.648,-178.187,10.219,149.552
C06986=1123.749,277.820,-73.618,-178.190,10.216,149.553
C06987=1123.754,277.572,-73.588,-178.193,10.214,149.553
C06988=1123.757,277.323,-73.557,-178.196,10.211,149.553
C06989=1123.761,277.076,-73.527,-178.199,10.208,149.553
C06990=1123.766,276.827,-73.497,-178.202,10.206,149.553
C06991=1123.770,276.579,-73.468,-178.205,10.203,149.553
C06992=1123.774,276.331,-73.438,-178.209,10.199,149.554
C06993=1123.779,276.083,-73.408,-178.212,10.197,149.554
C06994=1123.782,275.835,-73.377,-178.215,10.194,149.554
C06995=1123.787,275.587,-73.348,-178.218,10.192,149.554
C06996=1123.791,275.339,-73.318,-178.221,10.189,149.554
C06997=1123.795,275.090,-73.287,-178.225,10.186,149.554
C06998=1123.799,274.841,-73.258,-178.227,10.184,149.554
C06999=1123.803,274.594,-73.228,-178.230,10.181,149.555
C07000=1123.807,274.346,-73.198,-178.233,10.178,149.555
C07001=1123.812,274.098,-73.168,-178.237,10.176,149.555
C07002=1123.816,273.849,-73.138,-178.240,10.173,149.555
C07003=1123.820,273.601,-73.109,-178.243,10.170,149.555
C07004=1123.824,273.353,-73.079,-178.245,10.167,149.555
C07005=1123.828,273.105,-73.049,-178.248,10.165,149.555
C07006=1123.833,272.857,-73.019,-178.251,10.162,149.555
C07007=1123.837,272.608,-72.989,-178.254,10.159,149.556
C07008=1123.841,272.361,-72.959,-178.257,10.157,149.556
C07009=1123.845,272.112,-72.930,-178.260,10.154,149.556
C07010=1123.849,271.864,-72.900,-178.263,10.152,149.556
C07011=1123.854,271.616,-72.871,-178.266,10.149,149.556
C07012=1123.859,271.367,-72.841,-178.269,10.146,149.556
C07013=1123.862,271.120,-72.811,-178.272,10.144,149.556
C07014=1123.867,270.871,-72.781,-178.274,10.142,149.557
C07015=1123.871,270.623,-72.752,-178.277,10.139,149.557
C07016=1123.875,270.375,-72.722,-178.280,10.136,149.557
C07017=1123.879,270.127,-72.693,-178.283,10.133,149.557
C07018=1123.883,269.878,-72.663,-178.286,10.131,149.557
C07019=1123.888,269.630,-72.634,-178.288,10.129,149.557
C07020=1123.892,269.382,-72.605,-178.291,10.126,149.557
C07021=1123.896,269.133,-72.575,-178.294,10.123,149.557
C07022=1123.900,268.886,-72.545,-178.296,10.121,149.557
C07023=1123.905,268.637,-72.515,-178.299,10.118,149.557
C07024=1123.909,268.389,-72.485,-178.302,10.116,149.558
C07025=1123.913,268.141,-72.456,-178.304,10.114,149.558
C07026=1123.917,267.892,-72.427,-178.307,10.111,149.558
C07027=1123.921,267.679,-72.401,-178.309,10.109,149.558
C07028=1123.924,267.466,-72.376,-178.312,10.107,149.558
C07029=1123.928,267.252,-72.351,-178.314,10.105,149.558
C07030=1123.931,267.039,-72.326,-178.316,10.103,149.558
C07031=1123.935,266.825,-72.301,-178.319,10.101,149.558
C07032=1123.939,266.612,-72.275,-178.321,10.098,149.558
C07033=1123.943,266.399,-72.251,-178.323,10.096,149.558
C07034=1123.946,266.186,-72.225,-178.326,10.094,149.558
C07035=1123.951,265.938,-72.196,-178.328,10.092,149.559
C07036=1123.955,265.689,-72.167,-178.331,10.089,149.559
C07037=1123.959,265.441,-72.137,-178.333,10.087,149.559
C07038=1123.963,265.193,-72.108,-178.336,10.084,149.559
C07039=1123.968,264.944,-72.079,-178.338,10.082,149.559
C07040=1123.972,264.696,-72.049,-178.340,10.080,149.559
C07041=1123.976,264.447,-72.020,-178.343,10.077,149.559
C07042=1123.981,264.200,-71.991,-178.347,10.074,149.559
C07043=1123.985,263.951,-71.961,-178.351,10.071,149.560
C07044=1123.989,263.703,-71.932,-178.354,10.068,149.560
C07045=1123.994,263.454,-71.903,-178.358,10.065,149.560
C07046=1123.998,263.206,-71.874,-178.362,10.062,149.560
C07047=1124.001,262.958,-71.845,-178.365,10.059,149.560
C07048=1124.006,262.710,-71.817,-178.368,10.056,149.561
C07049=1124.010,262.462,-71.787,-178.372,10.053,149.561
C07050=1124.015,262.213,-71.758,-178.375,10.050,149.561
C07051=1124.019,261.965,-71.728,-178.379,10.047,149.561
C07052=1124.023,261.716,-71.699,-178.382,10.044,149.561
C07053=1124.027,261.469,-71.671,-178.386,10.041,149.562
C07054=1124.032,261.220,-71.642,-178.389,10.038,149.562
C07055=1124.036,260.972,-71.613,-178.392,10.036,149.562
C07056=1124.040,260.724,-71.583,-178.396,10.032,149.562
C07057=1124.045,260.476,-71.556,-178.399,10.030,149.562
C07058=1124.049,260.227,-71.526,-178.402,10.026,149.562
C07059=1124.053,259.978,-71.497,-178.405,10.023,149.562
C07060=1124.057,259.730,-71.468,-178.408,10.021,149.562
C07061=1124.062,259.482,-71.440,-178.411,10.018,149.563
C07062=1124.066,259.234,-71.411,-178.415,10.014,149.563
C07063=1124.070,258.985,-71.382,-178.418,10.011,149.563
C07064=1124.074,258.737,-71.353,-178.421,10.009,149.563
C07065=1124.079,258.489,-71.325,-178.423,10.006,149.563
C07066=1124.083,258.241,-71.295,-178.426,10.003,149.563
C07067=1124.087,257.992,-71.267,-178.430,10.000,149.563
C07068=1124.091,257.744,-71.238,-178.433,9.997,149.563
C07069=1124.096,257.496,-71.209,-178.436,9.994,149.563
C07070=1124.100,257.248,-71.180,-178.439,9.991,149.563
C07071=1124.104,256.999,-71.152,-178.442,9.989,149.564
C07072=1124.108,256.751,-71.124,-178.445,9.986,149.564
C07073=1124.113,256.503,-71.094,-178.447,9.983,149.564
C07074=1124.117,256.254,-71.066,-178.450,9.980,149.564
C07075=1124.121,256.006,-71.038,-178.453,9.977,149.564
C07076=1124.126,255.758,-71.009,-178.453,9.976,149.564
C07077=1124.129,255.509,-70.980,-178.454,9.975,149.563
C07078=1124.134,255.261,-70.952,-178.454,9.974,149.563
C07079=1124.139,255.013,-70.923,-178.455,9.972,149.563
C07080=1124.142,254.764,-70.894,-178.455,9.971,149.563
C07081=1124.147,254.516,-70.866,-178.456,9.969,149.563
C07082=1124.151,254.267,-70.838,-178.457,9.968,149.563
C07083=1124.155,254.054,-70.813,-178.459,9.966,149.563
C07084=1124.159,253.841,-70.789,-178.459,9.965,149.563
C07085=1124.162,253.628,-70.764,-178.461,9.963,149.563
C07086=1124.166,253.413,-70.740,-178.463,9.962,149.563
C07087=1124.170,253.200,-70.714,-178.464,9.960,149.563
C07088=1124.174,252.987,-70.690,-178.466,9.958,149.563
C07089=1124.177,252.773,-70.666,-178.468,9.957,149.563
C07090=1124.181,252.560,-70.641,-178.470,9.955,149.563
C07091=1124.186,252.311,-70.613,-178.473,9.952,149.563
C07092=1124.190,252.063,-70.585,-178.476,9.950,149.563
C07093=1124.194,251.815,-70.555,-178.479,9.947,149.563
C07094=1124.198,251.567,-70.527,-178.483,9.944,149.564
C07095=1124.203,251.318,-70.499,-178.486,9.942,149.564
C07096=1124.207,251.070,-70.471,-178.490,9.939,149.564
C07097=1124.211,250.821,-70.443,-178.493,9.936,149.564
C07098=1124.215,250.572,-70.414,-178.497,9.933,149.565
C07099=1124.219,250.325,-70.386,-178.501,9.929,149.565
C07100=1124.224,250.076,-70.358,-178.506,9.926,149.565
C07101=1124.228,249.828,-70.330,-178.511,9.922,149.566
C07102=1124.233,249.580,-70.300,-178.515,9.918,149.566
C07103=1124.237,249.332,-70.273,-178.520,9.915,149.566
C07104=1124.241,249.083,-70.244,-178.525,9.911,149.567
C07105=1124.245,248.834,-70.216,-178.530,9.906,149.567
C07106=1124.250,248.586,-70.189,-178.536,9.902,149.568
C07107=1124.254,248.337,-70.160,-178.542,9.898,149.568
C07108=1124.259,248.089,-70.132,-178.548,9.893,149.569
C07109=1124.263,247.841,-70.104,-178.554,9.888,149.569
C07110=1124.267,247.592,-70.076,-178.559,9.883,149.569
C07111=1124.271,247.345,-70.048,-178.564,9.880,149.570
C07112=1124.276,247.096,-70.020,-178.565,9.877,149.569
C07113=1124.280,246.847,-69.993,-178.566,9.875,149.569
C07114=1124.284,246.599,-69.964,-178.568,9.873,149.569
C07115=1124.288,246.351,-69.937,-178.570,9.870,149.569
C07116=1124.293,246.102,-69.908,-178.572,9.868,149.569
C07117=1124.297,245.853,-69.881,-178.573,9.866,149.569
C07118=1124.302,245.605,-69.853,-178.574,9.864,149.569
C07119=1124.306,245.357,-69.825,-178.576,9.861,149.569
C07120=1124.311,245.109,-69.797,-178.578,9.859,149.568
C07121=1124.315,244.860,-69.769,-178.580,9.857,149.568
C07122=1124.319,244.612,-69.741,-178.582,9.854,149.568
C07123=1124.323,244.363,-69.713,-178.584,9.852,149.568
C07124=1124.327,244.115,-69.686,-178.586,9.850,149.568
C07125=1124.332,243.867,-69.658,-178.588,9.847,149.568
C07126=1124.336,243.618,-69.630,-178.590,9.845,149.568
C07127=1124.341,243.369,-69.603,-178.592,9.843,149.568
C07128=1124.345,243.121,-69.574,-178.593,9.840,149.568
C07129=1124.349,242.873,-69.547,-178.595,9.838,149.568
C07130=1124.354,242.624,-69.520,-178.597,9.836,149.568
C07131=1124.357,242.376,-69.491,-178.600,9.834,149.568
C07132=1124.362,242.128,-69.464,-178.601,9.831,149.568
C07133=1124.367,241.878,-69.436,-178.603,9.829,149.568
C07134=1124.371,241.631,-69.408,-178.606,9.826,149.568
C07135=1124.376,241.382,-69.381,-178.608,9.824,149.568
C07136=1124.379,241.133,-69.353,-178.610,9.822,149.568
C07137=1124.384,240.886,-69.325,-178.612,9.820,149.568
C07138=1124.388,240.637,-69.298,-178.615,9.817,149.568
C07139=1124.391,240.423,-69.274,-178.617,9.815,149.568
C07140=1124.396,240.210,-69.250,-178.619,9.812,149.568
C07141=1124.399,239.996,-69.227,-178.621,9.811,149.568
C07142=1124.403,239.783,-69.203,-178.623,9.809,149.568
C07143=1124.407,239.569,-69.179,-178.625,9.807,149.568
C07144=1124.411,239.356,-69.155,-178.627,9.804,149.568
C07145=1124.414,239.141,-69.132,-178.629,9.802,149.568
C07146=1124.419,238.928,-69.108,-178.631,9.800,149.568
C07147=1124.422,238.679,-69.080,-178.634,9.797,149.568
C07148=1124.427,238.431,-69.053,-178.636,9.795,149.569
C07149=1124.431,238.183,-69.025,-178.639,9.792,149.569
C07150=1124.435,237.934,-68.998,-178.642,9.790,149.569
C07151=1124.440,237.685,-68.971,-178.644,9.788,149.569
C07152=1124.444,237.437,-68.943,-178.647,9.785,149.569
C07153=1124.449,237.188,-68.915,-178.650,9.782,149.569
C07154=1124.453,236.940,-68.888,-178.653,9.779,149.569
C07155=1124.458,236.692,-68.860,-178.655,9.777,149.569
C07156=1124.461,236.444,-68.834,-178.658,9.774,149.569
C07157=1124.466,236.194,-68.807,-178.661,9.771,149.569
C07158=1124.470,235.947,-68.779,-178.664,9.769,149.569
C07159=1124.475,235.698,-68.752,-178.667,9.766,149.570
C07160=1124.479,235.450,-68.725,-178.670,9.763,149.570
C07161=1124.483,235.201,-68.697,-178.672,9.760,149.570
C07162=1124.488,234.952,-68.669,-178.675,9.757,149.570
C07163=1124.492,234.704,-68.642,-178.678,9.755,149.570
C07164=1124.497,234.455,-68.615,-178.681,9.752,149.570
C07165=1124.501,234.207,-68.587,-178.684,9.749,149.570
C07166=1124.505,233.959,-68.561,-178.687,9.746,149.570
C07167=1124.509,233.710,-68.534,-178.690,9.744,149.570
C07168=1124.514,233.462,-68.507,-178.693,9.740,149.571
C07169=1124.519,233.213,-68.480,-178.696,9.737,149.571
C07170=1124.523,232.964,-68.452,-178.699,9.735,149.571
C07171=1124.527,232.716,-68.424,-178.702,9.732,149.571
C07172=1124.531,232.468,-68.398,-178.706,9.728,149.571
C07173=1124.536,232.219,-68.371,-178.709,9.726,149.571
C07174=1124.540,231.971,-68.344,-178.713,9.722,149.571
C07175=1124.544,231.722,-68.316,-178.716,9.720,149.572
C07176=1124.549,231.473,-68.289,-178.719,9.717,149.572
C07177=1124.553,231.225,-68.263,-178.722,9.713,149.572
C07178=1124.557,230.977,-68.236,-178.726,9.710,149.572
C07179=1124.562,230.728,-68.209,-178.729,9.707,149.572
C07180=1124.567,230.480,-68.182,-178.732,9.704,149.572
C07181=1124.571,230.231,-68.155,-178.736,9.700,149.572
C07182=1124.575,229.983,-68.128,-178.739,9.697,149.572
C07183=1124.579,229.734,-68.101,-178.742,9.694,149.573
C07184=1124.583,229.486,-68.074,-178.746,9.690,149.573
C07185=1124.588,229.237,-68.047,-178.750,9.687,149.573
C07186=1124.593,228.989,-68.020,-178.753,9.683,149.573
C07187=1124.597,228.740,-67.994,-178.756,9.681,149.573
C07188=1124.602,228.491,-67.967,-178.760,9.677,149.573
C07189=1124.606,228.243,-67.940,-178.763,9.673,149.573
C07190=1124.610,227.995,-67.914,-178.766,9.671,149.573
C07191=1124.615,227.746,-67.887,-178.770,9.667,149.573
C07192=1124.619,227.498,-67.860,-178.773,9.663,149.573
C07193=1124.623,227.249,-67.833,-178.776,9.661,149.574
C07194=1124.628,227.000,-67.807,-178.780,9.657,149.574
C07195=1124.631,226.786,-67.784,-178.782,9.654,149.574
C07196=1124.635,226.573,-67.761,-178.785,9.651,149.574
C07197=1124.639,226.360,-67.738,-178.788,9.648,149.574
C07198=1124.643,226.146,-67.715,-178.790,9.645,149.574
C07199=1124.646,225.932,-67.692,-178.792,9.643,149.574
C07200=1124.650,225.718,-67.669,-178.795,9.640,149.574
C07201=1124.654,225.504,-67.646,-178.798,9.637,149.574
C07202=1124.658,225.291,-67.624,-178.801,9.634,149.574
C07203=1124.663,225.042,-67.598,-178.803,9.631,149.574
C07204=1124.667,224.793,-67.571,-178.806,9.627,149.574
C07205=1124.671,224.545,-67.544,-178.809,9.625,149.574
C07206=1124.676,224.296,-67.518,-178.813,9.621,149.574
C07207=1124.680,224.048,-67.492,-178.815,9.618,149.574
C07208=1124.685,223.799,-67.465,-178.818,9.615,149.574
C07209=1124.689,223.551,-67.439,-178.821,9.611,149.574
C07210=1124.693,223.302,-67.412,-178.824,9.608,149.574
C07211=1124.698,223.053,-67.386,-178.826,9.605,149.574
C07212=1124.702,222.805,-67.359,-178.829,9.602,149.574
C07213=1124.707,222.556,-67.333,-178.832,9.598,149.574
C07214=1124.711,222.308,-67.307,-178.835,9.595,149.574
C07215=1124.715,222.059,-67.281,-178.837,9.592,149.574
C07216=1124.720,221.810,-67.255,-178.840,9.589,149.574
C07217=1124.724,221.562,-67.228,-178.842,9.586,149.573
C07218=1124.729,221.313,-67.202,-178.845,9.583,149.573
C07219=1124.733,221.065,-67.176,-178.848,9.580,149.573
C07220=1124.737,220.816,-67.150,-178.850,9.576,149.573
C07221=1124.742,220.568,-67.123,-178.853,9.573,149.573
C07222=1124.746,220.319,-67.097,-178.855,9.570,149.573
C07223=1124.751,220.070,-67.071,-178.858,9.567,149.573
C07224=1124.755,219.822,-67.044,-178.860,9.564,149.573
C07225=1124.759,219.573,-67.019,-178.862,9.561,149.573
C07226=1124.764,219.324,-66.993,-178.865,9.557,149.573
C07227=1124.768,219.077,-66.967,-178.867,9.554,149.573
C07228=1124.773,218.827,-66.940,-178.870,9.551,149.573
C07229=1124.777,218.579,-66.915,-178.872,9.548,149.573
C07230=1124.781,218.330,-66.888,-178.874,9.545,149.572
C07231=1124.785,218.082,-66.862,-178.876,9.542,149.572
C07232=1124.790,217.833,-66.836,-178.879,9.539,149.572
C07233=1124.795,217.584,-66.811,-178.881,9.536,149.572
C07234=1124.799,217.336,-66.784,-178.883,9.533,149.572
C07235=1124.803,217.087,-66.758,-178.885,9.530,149.572
C07236=1124.808,216.838,-66.732,-178.888,9.527,149.572
C07237=1124.813,216.590,-66.706,-178.889,9.524,149.571
C07238=1124.817,216.341,-66.681,-178.892,9.521,149.571
C07239=1124.821,216.093,-66.654,-178.894,9.518,149.571
C07240=1124.826,215.844,-66.629,-178.896,9.516,149.571
C07241=1124.830,215.596,-66.603,-178.898,9.512,149.571
C07242=1124.835,215.347,-66.577,-178.900,9.510,149.571
C07243=1124.840,215.098,-66.551,-178.902,9.507,149.571
C07244=1124.844,214.850,-66.525,-178.904,9.504,149.571
C07245=1124.848,214.601,-66.500,-178.906,9.502,149.570
C07246=1124.852,214.352,-66.474,-178.908,9.499,149.570
C07247=1124.856,214.104,-66.448,-178.910,9.496,149.570
C07248=1124.861,213.856,-66.422,-178.912,9.493,149.570
C07249=1124.866,213.607,-66.396,-178.914,9.490,149.570
C07250=1124.870,213.358,-66.370,-178.916,9.488,149.570
C07251=1124.874,213.144,-66.349,-178.918,9.485,149.570
C07252=1124.878,212.930,-66.326,-178.919,9.483,149.569
C07253=1124.881,212.716,-66.304,-178.920,9.481,149.569
C07254=1124.885,212.503,-66.281,-178.922,9.479,149.569
C07255=1124.889,212.289,-66.260,-178.924,9.476,149.569
C07256=1124.893,212.074,-66.238,-178.926,9.474,149.569
C07257=1124.897,211.861,-66.216,-178.928,9.471,149.569
C07258=1124.901,211.647,-66.194,-178.929,9.469,149.569
C07259=1124.905,211.398,-66.168,-178.931,9.467,149.569
C07260=1124.910,211.149,-66.142,-178.934,9.464,149.569
C07261=1124.914,210.901,-66.117,-178.936,9.461,149.569
C07262=1124.919,210.652,-66.091,-178.938,9.458,149.569
C07263=1124.923,210.403,-66.065,-178.940,9.456,149.569
C07264=1124.928,210.155,-66.040,-178.943,9.453,149.569
C07265=1124.932,209.907,-66.014,-178.945,9.450,149.569
C07266=1124.936,209.658,-65.988,-178.948,9.448,149.569
C07267=1124.941,209.410,-65.963,-178.949,9.445,149.569
C07268=1124.945,209.160,-65.938,-178.952,9.442,149.569
C07269=1124.950,208.911,-65.912,-178.954,9.439,149.569
C07270=1124.954,208.663,-65.887,-178.957,9.437,149.569
C07271=1124.959,208.414,-65.861,-178.959,9.434,149.569
C07272=1124.963,208.166,-65.835,-178.962,9.431,149.569
C07273=1124.968,207.918,-65.810,-178.964,9.429,149.569
C07274=1124.972,207.668,-65.785,-178.967,9.426,149.569
C07275=1124.977,207.419,-65.759,-178.970,9.423,149.569
C07276=1124.981,207.171,-65.734,-178.973,9.420,149.569
C07277=1124.986,206.922,-65.708,-178.974,9.418,149.569
C07278=1124.991,206.674,-65.683,-178.977,9.415,149.569
C07279=1124.995,206.425,-65.658,-178.980,9.412,149.569
C07280=1124.998,206.176,-65.632,-178.983,9.409,149.569
